LIN {X 0,Y 226.639,Z 302.23,A -85,B 0,C 180,E1 -22455.501,E2 -22455.501} C_VEL
LIN {X 0,Y 230.023,Z 288.136,A -85,B 0,C 180,E1 -22456.446,E2 -22456.446} C_VEL
LIN {X 0,Y 232.529,Z 273.347,A -85,B 0,C 180,E1 -22457.124,E2 -22457.124} C_VEL
LIN {X 0,Y 234.238,Z 254.152,A -85,B 0,C 180,E1 -22457.708,E2 -22457.708} C_VEL
LIN {X 0,Y 236.836,Z 218.214,A -85,B 0,C 180,E1 -22458.708,E2 -22458.708} C_VEL
LIN {X 0,Y 232.194,Z 207.283,A -85,B 0,C 180,E1 -22461.02,E2 -22461.02} C_VEL
LIN {X 0,Y 227.459,Z 197.713,A -85,B 0,C 180,E1 -22463.554,E2 -22463.554} C_VEL
LIN {X 0,Y 222.962,Z 189.346,A -85,B 0,C 180,E1 -22466.218,E2 -22466.218} C_VEL
LIN {X 0,Y 219.708,Z 183.706,A -85,B 0,C 180,E1 -22468.352,E2 -22468.352} C_VEL
LIN {X 0,Y 216.874,Z 179.005,A -85,B 0,C 180,E1 -22470.433,E2 -22470.433} C_VEL
LIN {X 0,Y 214.738,Z 175.538,A -85,B 0,C 180,E1 -22472.178,E2 -22472.178} C_VEL
LIN {X 0,Y 211.845,Z 170.966,A -85,B 0,C 180,E1 -22474.848,E2 -22474.848} C_VEL
LIN {X 0,Y 209.156,Z 167.545,A -85,B 0,C 180,E1 -22477.703,E2 -22477.703} C_VEL
LIN {X 0,Y 207.226,Z 164.238,A -85,B 0,C 180,E1 -22480.325,E2 -22480.325} C_VEL
LIN {X 0,Y 203.698,Z 160.294,A -85,B 0,C 180,E1 -22488.046,E2 -22488.046} C_VEL
LIN {X 0,Y 203.417,Z 158.582,A -85,B 0,C 180,E1 -22490.606,E2 -22490.606} C_VEL
LIN {X 0,Y 203.441,Z 158.596,A -85,B 0,C 180,E1 -22494.045,E2 -22494.045} C_VEL
LIN {X 0,Y 204.542,Z 161.074,A -85,B 0,C 180,E1 -22499.009,E2 -22499.009} C_VEL
LIN {X 0,Y 206.776,Z 163.712,A -85,B 0,C 180,E1 -22503.403,E2 -22503.403} C_VEL
LIN {X 0,Y 207.532,Z 164.297,A -85,B 0,C 180,E1 -22504.485,E2 -22504.485} C_VEL
LIN {X 0,Y 209.461,Z 167.504,A -85,B 0,C 180,E1 -22507.018,E2 -22507.018} C_VEL
LIN {X 0,Y 211.323,Z 169.48,A -85,B 0,C 180,E1 -22508.967,E2 -22508.967} C_VEL
LIN {X 0,Y 213.7,Z 172.996,A -85,B 0,C 180,E1 -22511.242,E2 -22511.242} C_VEL
LIN {X 0,Y 215.003,Z 174.469,A -85,B 0,C 180,E1 -22512.327,E2 -22512.327} C_VEL
LIN {X 0,Y 218.65,Z 179.753,A -85,B 0,C 180,E1 -22515.145,E2 -22515.145} C_VEL
LIN {X 0,Y 221.809,Z 184.298,A -85,B 0,C 180,E1 -22517.251,E2 -22517.251} C_VEL
LIN {X 0,Y 225.031,Z 189.073,A -85,B 0,C 180,E1 -22519.193,E2 -22519.193} C_VEL
LIN {X 0,Y 229.645,Z 196.427,A -85,B 0,C 180,E1 -22521.724,E2 -22521.724} C_VEL
LIN {X 0,Y 234.735,Z 206.452,A -85,B 0,C 180,E1 -22524.318,E2 -22524.318} C_VEL
LIN {X 0,Y 237.283,Z 212.078,A -85,B 0,C 180,E1 -22525.544,E2 -22525.544} C_VEL
LIN {X 0,Y 233.316,Z 263.334,A -85,B 0,C 180,E1 -22526.974,E2 -22526.974} C_VEL
LIN {X 0,Y 231.209,Z 277.512,A -85,B 0,C 180,E1 -22527.622,E2 -22527.622} C_VEL
LIN {X 0,Y 228.377,Z 290.64,A -85,B 0,C 180,E1 -22528.477,E2 -22528.477} C_VEL
LIN {X 0,Y 224.932,Z 303.341,A -85,B 0,C 180,E1 -22529.627,E2 -22529.627} C_VEL
LIN {X 0,Y 220.658,Z 316.029,A -85,B 0,C 180,E1 -22531.128,E2 -22531.128} C_VEL
LIN {X 0,Y 215.677,Z 328.153,A -85,B 0,C 180,E1 -22532.953,E2 -22532.953} C_VEL
LIN {X 0,Y 210.464,Z 339.178,A -85,B 0,C 180,E1 -22535.098,E2 -22535.098} C_VEL
LIN {X 0,Y 205.553,Z 348.32,A -85,B 0,C 180,E1 -22537.347,E2 -22537.347} C_VEL
LIN {X 0,Y 200.034,Z 357.449,A -85,B 0,C 180,E1 -22540.163,E2 -22540.163} C_VEL
LIN {X 0,Y 195.008,Z 365.073,A -85,B 0,C 180,E1 -22543.205,E2 -22543.205} C_VEL
LIN {X 0,Y 190.001,Z 372.031,A -85,B 0,C 180,E1 -22546.816,E2 -22546.816} C_VEL
LIN {X 0,Y 186.208,Z 376.82,A -85,B 0,C 180,E1 -22550.083,E2 -22550.083} C_VEL
LIN {X 0,Y 182.741,Z 380.951,A -85,B 0,C 180,E1 -22553.85,E2 -22553.85} C_VEL
LIN {X 0,Y 180.515,Z 383.439,A -85,B 0,C 180,E1 -22556.967,E2 -22556.967} C_VEL
LIN {X 0,Y 177.978,Z 385.836,A -85,B 0,C 180,E1 -22561.712,E2 -22561.712} C_VEL
LIN {X 0,Y 176.489,Z 386.756,A -85,B 0,C 180,E1 -22566.53,E2 -22566.53} C_VEL
LIN {X 0,Y 175.717,Z 386.244,A -85,B 0,C 180,E1 -22571.336,E2 -22571.336} C_VEL
LIN {X 0,Y 175.641,Z 385.441,A -85,B 0,C 180,E1 -22573.772,E2 -22573.772} C_VEL
LIN {X 0,Y 175.765,Z 382.819,A -85,B 0,C 180,E1 -22578.464,E2 -22578.464} C_VEL
LIN {X 0,Y 176.339,Z 379.84,A -85,B 0,C 180,E1 -22581.978,E2 -22581.978} C_VEL
LIN {X 0,Y 177.183,Z 376.025,A -85,B 0,C 180,E1 -22585.447,E2 -22585.447} C_VEL
LIN {X 0,Y 178.317,Z 371.31,A -85,B 0,C 180,E1 -22588.868,E2 -22588.868} C_VEL
LIN {X 0,Y 180.274,Z 364.443,A -85,B 0,C 180,E1 -22592.79,E2 -22592.79} C_VEL
LIN {X 0,Y 182.883,Z 355.918,A -85,B 0,C 180,E1 -22596.617,E2 -22596.617} C_VEL
LIN {X 0,Y 185.69,Z 346.926,A -85,B 0,C 180,E1 -22599.834,E2 -22599.834} C_VEL
LIN {X 0,Y 188.154,Z 338.243,A -85,B 0,C 180,E1 -22602.399,E2 -22602.399} C_VEL
LIN {X 0,Y 190.884,Z 328.903,A -85,B 0,C 180,E1 -22604.659,E2 -22604.659} C_VEL
LIN {X 0,Y 193.794,Z 317.727,A -85,B 0,C 180,E1 -22606.862,E2 -22606.862} C_VEL
LIN {X 0,Y 196.61,Z 305.55,A -85,B 0,C 180,E1 -22608.763,E2 -22608.763} C_VEL
LIN {X 0,Y 199.157,Z 292.089,A -85,B 0,C 180,E1 -22610.391,E2 -22610.391} C_VEL
LIN {X 0,Y 201.213,Z 278.05,A -85,B 0,C 180,E1 -22611.646,E2 -22611.646} C_VEL
LIN {X 0,Y 202.695,Z 263.821,A -85,B 0,C 180,E1 -22612.518,E2 -22612.518} C_VEL
LIN {X 0,Y 204.368,Z 237.316,A -85,B 0,C 180,E1 -22613.431,E2 -22613.431} C_VEL
LIN {X 0,Y 207.071,Z 187.142,A -85,B 0,C 180,E1 -22615.036,E2 -22615.036} C_VEL
LIN {X 0,Y 202.861,Z 176.015,A -85,B 0,C 180,E1 -22616.361,E2 -22616.361} C_VEL
LIN {X 0,Y 196.456,Z 163.46,A -85,B 0,C 180,E1 -22618.321,E2 -22618.321} C_VEL
LIN {X 0,Y 188.904,Z 150.475,A -85,B 0,C 180,E1 -22620.783,E2 -22620.783} C_VEL
LIN {X 0,Y 183.421,Z 142.139,A -85,B 0,C 180,E1 -22622.704,E2 -22622.704} C_VEL
LIN {X 0,Y 180.927,Z 138.404,A -85,B 0,C 180,E1 -22623.626,E2 -22623.626} C_VEL
LIN {X 0,Y 179.099,Z 136.063,A -85,B 0,C 180,E1 -22624.304,E2 -22624.304} C_VEL
LIN {X 0,Y 178.464,Z 133.88,A -85,B 0,C 180,E1 -22624.658,E2 -22624.658} C_VEL
LIN {X 0,Y 178.477,Z 133.875,A -85,B 0,C 180,E1 -22629.049,E2 -22629.049} C_VEL
LIN {X 0,Y 178.494,Z 133.859,A -85,B 0,C 180,E1 -22632.013,E2 -22632.013} C_VEL
LIN {X 0,Y 178.504,Z 133.854,A -85,B 0,C 180,E1 -22635.123,E2 -22635.123} C_VEL
LIN {X 0,Y 178.493,Z 133.87,A -85,B 0,C 180,E1 -22638.421,E2 -22638.421} C_VEL
LIN {X 0,Y 178.444,Z 133.86,A -85,B 0,C 180,E1 -22643.799,E2 -22643.799} C_VEL
LIN {X 0,Y 178.466,Z 133.878,A -85,B 0,C 180,E1 -22646.553,E2 -22646.553} C_VEL
LIN {X 0,Y 178.499,Z 133.842,A -85,B 0,C 180,E1 -22650.013,E2 -22650.013} C_VEL
LIN {X 0,Y 178.525,Z 133.862,A -85,B 0,C 180,E1 -22654.875,E2 -22654.875} C_VEL
LIN {X 0,Y 178.638,Z 133.852,A -85,B 0,C 180,E1 -22660.761,E2 -22660.761} C_VEL
LIN {X 0,Y 178.663,Z 133.849,A -85,B 0,C 180,E1 -22664.025,E2 -22664.025} C_VEL
LIN {X 0,Y 178.88,Z 133.825,A -85,B 0,C 180,E1 -22669.161,E2 -22669.161} C_VEL
LIN {X 0,Y 178.918,Z 133.782,A -85,B 0,C 180,E1 -22673.24,E2 -22673.24} C_VEL
LIN {X 0,Y 179.146,Z 133.788,A -85,B 0,C 180,E1 -22677.759,E2 -22677.759} C_VEL
LIN {X 0,Y 179.363,Z 133.764,A -85,B 0,C 180,E1 -22680.007,E2 -22680.007} C_VEL
LIN {X 0,Y 178.863,Z 133.791,A -85,B 0,C 180,E1 -22684.515,E2 -22684.515} C_VEL
LIN {X 0,Y 178.953,Z 133.817,A -85,B 0,C 180,E1 -22689.045,E2 -22689.045} C_VEL
LIN {X 0,Y 178.682,Z 133.85,A -85,B 0,C 180,E1 -22693.657,E2 -22693.657} C_VEL
LIN {X 0,Y 178.647,Z 133.853,A -85,B 0,C 180,E1 -22698.351,E2 -22698.351} C_VEL
LIN {X 0,Y 178.51,Z 133.872,A -85,B 0,C 180,E1 -22703.192,E2 -22703.192} C_VEL
LIN {X 0,Y 178.487,Z 133.863,A -85,B 0,C 180,E1 -22708.204,E2 -22708.204} C_VEL
LIN {X 0,Y 178.479,Z 133.872,A -85,B 0,C 180,E1 -22710.798,E2 -22710.798} C_VEL
LIN {X 0,Y 178.486,Z 133.875,A -85,B 0,C 180,E1 -22714.226,E2 -22714.226} C_VEL
LIN {X 0,Y 178.411,Z 134.02,A -85,B 0,C 180,E1 -22719,E2 -22719} C_VEL
LIN {X 0,Y 179.403,Z 136.688,A -85,B 0,C 180,E1 -22719.454,E2 -22719.454} C_VEL
LIN {X 0,Y 181.505,Z 139.246,A -85,B 0,C 180,E1 -22720.224,E2 -22720.224} C_VEL
LIN {X 0,Y 183.847,Z 142.743,A -85,B 0,C 180,E1 -22721.083,E2 -22721.083} C_VEL
LIN {X 0,Y 187.701,Z 149.384,A -85,B 0,C 180,E1 -22722.472,E2 -22722.472} C_VEL
LIN {X 0,Y 194.053,Z 161.878,A -85,B 0,C 180,E1 -22724.674,E2 -22724.674} C_VEL
LIN {X 0,Y 199.515,Z 174.348,A -85,B 0,C 180,E1 -22726.489,E2 -22726.489} C_VEL
LIN {X 0,Y 206.104,Z 192.069,A -85,B 0,C 180,E1 -22728.614,E2 -22728.614} C_VEL
LIN {X 0,Y 206.691,Z 198.413,A -85,B 0,C 180,E1 -22728.996,E2 -22728.996} C_VEL
LIN {X 0,Y 204.55,Z 238.997,A -85,B 0,C 180,E1 -22730.302,E2 -22730.302} C_VEL
LIN {X 0,Y 203.682,Z 244.836,A -85,B 0,C 180,E1 -22730.383,E2 -22730.383} C_VEL
LIN {X 0,Y 197.843,Z 263.771,A -85,B 0,C 180,E1 -22730.101,E2 -22730.101} C_VEL
LIN {X 0,Y 196.93,Z 269.591,A -85,B 0,C 180,E1 -22730.223,E2 -22730.223} C_VEL
LIN {X 0,Y 195.435,Z 283.943,A -85,B 0,C 180,E1 -22731.004,E2 -22731.004} C_VEL
LIN {X 0,Y 193.223,Z 297.885,A -85,B 0,C 180,E1 -22732.14,E2 -22732.14} C_VEL
LIN {X 0,Y 190.752,Z 310.484,A -85,B 0,C 180,E1 -22733.555,E2 -22733.555} C_VEL
LIN {X 0,Y 187.973,Z 322.176,A -85,B 0,C 180,E1 -22735.243,E2 -22735.243} C_VEL
LIN {X 0,Y 184.761,Z 334.344,A -85,B 0,C 180,E1 -22737.505,E2 -22737.505} C_VEL
LIN {X 0,Y 182.676,Z 341.22,A -85,B 0,C 180,E1 -22739.035,E2 -22739.035} C_VEL
LIN {X 0,Y 179.29,Z 352.041,A -85,B 0,C 180,E1 -22741.944,E2 -22741.944} C_VEL
LIN {X 0,Y 176.224,Z 361.794,A -85,B 0,C 180,E1 -22745.248,E2 -22745.248} C_VEL
LIN {X 0,Y 173.711,Z 369.855,A -85,B 0,C 180,E1 -22748.65,E2 -22748.65} C_VEL
LIN {X 0,Y 171.794,Z 376.544,A -85,B 0,C 180,E1 -22752.136,E2 -22752.136} C_VEL
LIN {X 0,Y 170.316,Z 382.067,A -85,B 0,C 180,E1 -22755.669,E2 -22755.669} C_VEL
LIN {X 0,Y 169.282,Z 387.851,A -85,B 0,C 180,E1 -22760.444,E2 -22760.444} C_VEL
LIN {X 0,Y 168.89,Z 392.01,A -85,B 0,C 180,E1 -22765.229,E2 -22765.229} C_VEL
LIN {X 0,Y 169.024,Z 394.686,A -85,B 0,C 180,E1 -22770.003,E2 -22770.003} C_VEL
LIN {X 0,Y 168.891,Z 395.944,A -85,B 0,C 180,E1 -22774.777,E2 -22774.777} C_VEL
LIN {X 0,Y 169.339,Z 395.878,A -85,B 0,C 180,E1 -22779.559,E2 -22779.559} C_VEL
LIN {X 0,Y 170.625,Z 394.512,A -85,B 0,C 180,E1 -22784.312,E2 -22784.312} C_VEL
LIN {X 0,Y 173.086,Z 391.826,A -85,B 0,C 180,E1 -22788.959,E2 -22788.959} C_VEL
LIN {X 0,Y 176.47,Z 387.752,A -85,B 0,C 180,E1 -22793.472,E2 -22793.472} C_VEL
LIN {X 0,Y 180.936,Z 382.174,A -85,B 0,C 180,E1 -22797.785,E2 -22797.785} C_VEL
LIN {X 0,Y 186.475,Z 374.921,A -85,B 0,C 180,E1 -22801.85,E2 -22801.85} C_VEL
LIN {X 0,Y 192.081,Z 366.957,A -85,B 0,C 180,E1 -22805.192,E2 -22805.192} C_VEL
LIN {X 0,Y 197.505,Z 358.65,A -85,B 0,C 180,E1 -22807.87,E2 -22807.87} C_VEL
LIN {X 0,Y 203.298,Z 348.508,A -85,B 0,C 180,E1 -22810.481,E2 -22810.481} C_VEL
LIN {X 0,Y 208.899,Z 337.644,A -85,B 0,C 180,E1 -22812.618,E2 -22812.618} C_VEL
LIN {X 0,Y 214.296,Z 325.305,A -85,B 0,C 180,E1 -22814.511,E2 -22814.511} C_VEL
LIN {X 0,Y 218.855,Z 313.118,A -85,B 0,C 180,E1 -22815.936,E2 -22815.936} C_VEL
LIN {X 0,Y 223.004,Z 299.599,A -85,B 0,C 180,E1 -22817.119,E2 -22817.119} C_VEL
LIN {X 0,Y 226.211,Z 286.174,A -85,B 0,C 180,E1 -22817.967,E2 -22817.967} C_VEL
LIN {X 0,Y 228.574,Z 271.708,A -85,B 0,C 180,E1 -22818.618,E2 -22818.618} C_VEL
LIN {X 0,Y 231.009,Z 242.939,A -85,B 0,C 180,E1 -22819.448,E2 -22819.448} C_VEL
LIN {X 0,Y 232.645,Z 221.01,A -85,B 0,C 180,E1 -22820.066,E2 -22820.066} C_VEL
LIN {X 0,Y 228.436,Z 211.057,A -85,B 0,C 180,E1 -22822.307,E2 -22822.307} C_VEL
LIN {X 0,Y 224.376,Z 202.623,A -85,B 0,C 180,E1 -22824.627,E2 -22824.627} C_VEL
LIN {X 0,Y 220.353,Z 194.856,A -85,B 0,C 180,E1 -22827.16,E2 -22827.16} C_VEL
LIN {X 0,Y 216.306,Z 187.516,A -85,B 0,C 180,E1 -22830.06,E2 -22830.06} C_VEL
LIN {X 0,Y 212.889,Z 181.881,A -85,B 0,C 180,E1 -22832.9,E2 -22832.9} C_VEL
LIN {X 0,Y 209.749,Z 176.823,A -85,B 0,C 180,E1 -22835.99,E2 -22835.99} C_VEL
LIN {X 0,Y 206.06,Z 171.29,A -85,B 0,C 180,E1 -22840.669,E2 -22840.669} C_VEL
LIN {X 0,Y 205.511,Z 170.742,A -85,B 0,C 180,E1 -22841.528,E2 -22841.528} C_VEL
LIN {X 0,Y 202.644,Z 166.883,A -85,B 0,C 180,E1 -22848.997,E2 -22848.997} C_VEL
LIN {X 0,Y 202.501,Z 165.535,A -85,B 0,C 180,E1 -22851.124,E2 -22851.124} C_VEL
LIN {X 0,Y 202.572,Z 165.825,A -85,B 0,C 180,E1 -22854.283,E2 -22854.283} C_VEL
LIN {X 0,Y 203.553,Z 168.062,A -85,B 0,C 180,E1 -22858.757,E2 -22858.757} C_VEL
LIN {X 0,Y 205.721,Z 170.676,A -85,B 0,C 180,E1 -22863.176,E2 -22863.176} C_VEL
LIN {X 0,Y 206.358,Z 171.324,A -85,B 0,C 180,E1 -22864.144,E2 -22864.144} C_VEL
LIN {X 0,Y 208.446,Z 174.671,A -85,B 0,C 180,E1 -22866.938,E2 -22866.938} C_VEL
LIN {X 0,Y 209.825,Z 176.191,A -85,B 0,C 180,E1 -22868.426,E2 -22868.426} C_VEL
LIN {X 0,Y 212.302,Z 179.809,A -85,B 0,C 180,E1 -22870.871,E2 -22870.871} C_VEL
LIN {X 0,Y 213.441,Z 181.322,A -85,B 0,C 180,E1 -22871.869,E2 -22871.869} C_VEL
LIN {X 0,Y 216.66,Z 186.081,A -85,B 0,C 180,E1 -22874.458,E2 -22874.458} C_VEL
LIN {X 0,Y 219.723,Z 190.648,A -85,B 0,C 180,E1 -22876.611,E2 -22876.611} C_VEL
LIN {X 0,Y 223.585,Z 196.497,A -85,B 0,C 180,E1 -22879.006,E2 -22879.006} C_VEL
LIN {X 0,Y 227.202,Z 202.77,A -85,B 0,C 180,E1 -22881.074,E2 -22881.074} C_VEL
LIN {X 0,Y 231.568,Z 211.613,A -85,B 0,C 180,E1 -22883.406,E2 -22883.406} C_VEL
LIN {X 0,Y 233.113,Z 215.025,A -85,B 0,C 180,E1 -22884.192,E2 -22884.192} C_VEL
LIN {X 0,Y 229.221,Z 263.339,A -85,B 0,C 180,E1 -22885.54,E2 -22885.54} C_VEL
LIN {X 0,Y 227.09,Z 277.278,A -85,B 0,C 180,E1 -22886.165,E2 -22886.165} C_VEL
LIN {X 0,Y 223.982,Z 291.266,A -85,B 0,C 180,E1 -22887.08,E2 -22887.08} C_VEL
LIN {X 0,Y 220.076,Z 304.924,A -85,B 0,C 180,E1 -22888.339,E2 -22888.339} C_VEL
LIN {X 0,Y 215.7,Z 317.206,A -85,B 0,C 180,E1 -22889.826,E2 -22889.826} C_VEL
LIN {X 0,Y 210.567,Z 329.156,A -85,B 0,C 180,E1 -22891.664,E2 -22891.664} C_VEL
LIN {X 0,Y 205.077,Z 340.216,A -85,B 0,C 180,E1 -22893.864,E2 -22893.864} C_VEL
LIN {X 0,Y 199.376,Z 350.204,A -85,B 0,C 180,E1 -22896.415,E2 -22896.415} C_VEL
LIN {X 0,Y 193.426,Z 359.414,A -85,B 0,C 180,E1 -22899.453,E2 -22899.453} C_VEL
LIN {X 0,Y 187.543,Z 367.661,A -85,B 0,C 180,E1 -22903.047,E2 -22903.047} C_VEL
LIN {X 0,Y 183.113,Z 373.348,A -85,B 0,C 180,E1 -22906.298,E2 -22906.298} C_VEL
LIN {X 0,Y 179.21,Z 377.935,A -85,B 0,C 180,E1 -22909.675,E2 -22909.675} C_VEL
LIN {X 0,Y 175.978,Z 381.516,A -85,B 0,C 180,E1 -22913.194,E2 -22913.194} C_VEL
LIN {X 0,Y 174.174,Z 383.378,A -85,B 0,C 180,E1 -22915.601,E2 -22915.601} C_VEL
LIN {X 0,Y 171.368,Z 385.895,A -85,B 0,C 180,E1 -22920.515,E2 -22920.515} C_VEL
LIN {X 0,Y 169.591,Z 386.933,A -85,B 0,C 180,E1 -22925.514,E2 -22925.514} C_VEL
LIN {X 0,Y 168.69,Z 386.534,A -85,B 0,C 180,E1 -22930.528,E2 -22930.528} C_VEL
LIN {X 0,Y 168.56,Z 385.64,A -85,B 0,C 180,E1 -22933.496,E2 -22933.496} C_VEL
LIN {X 0,Y 168.611,Z 383.286,A -85,B 0,C 180,E1 -22937.967,E2 -22937.967} C_VEL
LIN {X 0,Y 169.155,Z 380.413,A -85,B 0,C 180,E1 -22941.635,E2 -22941.635} C_VEL
LIN {X 0,Y 170.001,Z 376.719,A -85,B 0,C 180,E1 -22945.254,E2 -22945.254} C_VEL
LIN {X 0,Y 171.156,Z 372.089,A -85,B 0,C 180,E1 -22948.82,E2 -22948.82} C_VEL
LIN {X 0,Y 173.133,Z 365.392,A -85,B 0,C 180,E1 -22952.905,E2 -22952.905} C_VEL
LIN {X 0,Y 175.802,Z 357.048,A -85,B 0,C 180,E1 -22956.885,E2 -22956.885} C_VEL
LIN {X 0,Y 178.897,Z 347.578,A -85,B 0,C 180,E1 -22960.443,E2 -22960.443} C_VEL
LIN {X 0,Y 181.767,Z 337.828,A -85,B 0,C 180,E1 -22963.411,E2 -22963.411} C_VEL
LIN {X 0,Y 184.659,Z 328.358,A -85,B 0,C 180,E1 -22965.731,E2 -22965.731} C_VEL
LIN {X 0,Y 187.72,Z 317.02,A -85,B 0,C 180,E1 -22967.988,E2 -22967.988} C_VEL
LIN {X 0,Y 190.631,Z 304.642,A -85,B 0,C 180,E1 -22969.936,E2 -22969.936} C_VEL
LIN {X 0,Y 193.322,Z 290.861,A -85,B 0,C 180,E1 -22971.594,E2 -22971.594} C_VEL
LIN {X 0,Y 195.335,Z 277.112,A -85,B 0,C 180,E1 -22972.821,E2 -22972.821} C_VEL
LIN {X 0,Y 196.839,Z 262.88,A -85,B 0,C 180,E1 -22973.68,E2 -22973.68} C_VEL
LIN {X 0,Y 200.447,Z 203.666,A -85,B 0,C 180,E1 -22975.643,E2 -22975.643} C_VEL
LIN {X 0,Y 201.212,Z 188.949,A -85,B 0,C 180,E1 -22976.135,E2 -22976.135} C_VEL
LIN {X 0,Y 197.357,Z 178.875,A -85,B 0,C 180,E1 -22977.409,E2 -22977.409} C_VEL
LIN {X 0,Y 191.075,Z 166.594,A -85,B 0,C 180,E1 -22979.443,E2 -22979.443} C_VEL
LIN {X 0,Y 184.097,Z 154.645,A -85,B 0,C 180,E1 -22981.856,E2 -22981.856} C_VEL
LIN {X 0,Y 177.132,Z 143.849,A -85,B 0,C 180,E1 -22984.475,E2 -22984.475} C_VEL
LIN {X 0,Y 174.957,Z 140.891,A -85,B 0,C 180,E1 -22985.334,E2 -22985.334} C_VEL
LIN {X 0,Y 174.114,Z 139.492,A -85,B 0,C 180,E1 -22985.691,E2 -22985.691} C_VEL
LIN {X 0,Y 172.15,Z 137.141,A -85,B 0,C 180,E1 -22986.492,E2 -22986.492} C_VEL
LIN {X 0,Y 171.41,Z 134.76,A -85,B 0,C 180,E1 -22986.954,E2 -22986.954} C_VEL
LIN {X 0,Y 171.434,Z 134.733,A -85,B 0,C 180,E1 -22992.46,E2 -22992.46} C_VEL
LIN {X 0,Y 171.432,Z 134.753,A -85,B 0,C 180,E1 -22997.549,E2 -22997.549} C_VEL
LIN {X 0,Y 171.417,Z 134.721,A -85,B 0,C 180,E1 -23002.06,E2 -23002.06} C_VEL
LIN {X 0,Y 171.395,Z 134.752,A -85,B 0,C 180,E1 -23007.798,E2 -23007.798} C_VEL
LIN {X 0,Y 171.426,Z 134.718,A -85,B 0,C 180,E1 -23010.54,E2 -23010.54} C_VEL
LIN {X 0,Y 171.453,Z 134.75,A -85,B 0,C 180,E1 -23015.81,E2 -23015.81} C_VEL
LIN {X 0,Y 171.594,Z 134.73,A -85,B 0,C 180,E1 -23020.882,E2 -23020.882} C_VEL
LIN {X 0,Y 171.599,Z 134.724,A -85,B 0,C 180,E1 -23025.783,E2 -23025.783} C_VEL
LIN {X 0,Y 171.894,Z 134.682,A -85,B 0,C 180,E1 -23030.596,E2 -23030.596} C_VEL
LIN {X 0,Y 171.814,Z 134.673,A -85,B 0,C 180,E1 -23035.315,E2 -23035.315} C_VEL
LIN {X 0,Y 172.325,Z 134.641,A -85,B 0,C 180,E1 -23040.008,E2 -23040.008} C_VEL
LIN {X 0,Y 171.812,Z 134.668,A -85,B 0,C 180,E1 -23044.7,E2 -23044.7} C_VEL
LIN {X 0,Y 171.883,Z 134.7,A -85,B 0,C 180,E1 -23049.421,E2 -23049.421} C_VEL
LIN {X 0,Y 171.605,Z 134.733,A -85,B 0,C 180,E1 -23054.232,E2 -23054.232} C_VEL
LIN {X 0,Y 171.542,Z 134.742,A -85,B 0,C 180,E1 -23059.57,E2 -23059.57} C_VEL
LIN {X 0,Y 171.469,Z 134.749,A -85,B 0,C 180,E1 -23065.624,E2 -23065.624} C_VEL
LIN {X 0,Y 171.442,Z 134.75,A -85,B 0,C 180,E1 -23070.594,E2 -23070.594} C_VEL
LIN {X 0,Y 171.391,Z 134.759,A -85,B 0,C 180,E1 -23076.674,E2 -23076.674} C_VEL
LIN {X 0,Y 172.273,Z 137.408,A -85,B 0,C 180,E1 -23077.185,E2 -23077.185} C_VEL
LIN {X 0,Y 174.601,Z 140.281,A -85,B 0,C 180,E1 -23078.138,E2 -23078.138} C_VEL
LIN {X 0,Y 176.859,Z 143.654,A -85,B 0,C 180,E1 -23079.056,E2 -23079.056} C_VEL
LIN {X 0,Y 181.273,Z 150.337,A -85,B 0,C 180,E1 -23080.752,E2 -23080.752} C_VEL
LIN {X 0,Y 187.137,Z 161.585,A -85,B 0,C 180,E1 -23082.94,E2 -23082.94} C_VEL
LIN {X 0,Y 193.134,Z 174.722,A -85,B 0,C 180,E1 -23085.065,E2 -23085.065} C_VEL
LIN {X 0,Y 199.773,Z 192.505,A -85,B 0,C 180,E1 -23087.355,E2 -23087.355} C_VEL
LIN {X 0,Y 200.577,Z 195.66,A -85,B 0,C 180,E1 -23087.662,E2 -23087.662} C_VEL
LIN {X 0,Y 200.829,Z 199.802,A -85,B 0,C 180,E1 -23087.896,E2 -23087.896} C_VEL
LIN {X 0,Y 196.93,Z 269.591,A -85,B 0,C 180,E1 -23090.223,E2 -23090.223} C_VEL
LIN {X 0,Y 195.922,Z 275.384,A -85,B 0,C 180,E1 -23090.386,E2 -23090.386} C_VEL
LIN {X 0,Y 192.455,Z 284.667,A -85,B 0,C 180,E1 -23090.492,E2 -23090.492} C_VEL
LIN {X 0,Y 188.566,Z 293.775,A -85,B 0,C 180,E1 -23090.753,E2 -23090.753} C_VEL
LIN {X 0,Y 186.912,Z 299.299,A -85,B 0,C 180,E1 -23091.168,E2 -23091.168} C_VEL
LIN {X 0,Y 184.166,Z 312.3,A -85,B 0,C 180,E1 -23092.717,E2 -23092.717} C_VEL
LIN {X 0,Y 181.138,Z 324.295,A -85,B 0,C 180,E1 -23094.576,E2 -23094.576} C_VEL
LIN {X 0,Y 178.389,Z 334.306,A -85,B 0,C 180,E1 -23096.53,E2 -23096.53} C_VEL
LIN {X 0,Y 176.213,Z 341.167,A -85,B 0,C 180,E1 -23098.103,E2 -23098.103} C_VEL
LIN {X 0,Y 172.993,Z 351.059,A -85,B 0,C 180,E1 -23100.827,E2 -23100.827} C_VEL
LIN {X 0,Y 169.732,Z 360.942,A -85,B 0,C 180,E1 -23104.233,E2 -23104.233} C_VEL
LIN {X 0,Y 166.992,Z 369.253,A -85,B 0,C 180,E1 -23107.819,E2 -23107.819} C_VEL
LIN {X 0,Y 164.703,Z 376.93,A -85,B 0,C 180,E1 -23111.983,E2 -23111.983} C_VEL
LIN {X 0,Y 163.006,Z 383.156,A -85,B 0,C 180,E1 -23116.286,E2 -23116.286} C_VEL
LIN {X 0,Y 162.227,Z 387.382,A -85,B 0,C 180,E1 -23120.025,E2 -23120.025} C_VEL
LIN {X 0,Y 161.946,Z 389.695,A -85,B 0,C 180,E1 -23122.523,E2 -23122.523} C_VEL
LIN {X 0,Y 161.814,Z 393.172,A -85,B 0,C 180,E1 -23127.514,E2 -23127.514} C_VEL
LIN {X 0,Y 161.934,Z 394.368,A -85,B 0,C 180,E1 -23130.004,E2 -23130.004} C_VEL
LIN {X 0,Y 161.81,Z 395.698,A -85,B 0,C 180,E1 -23134.987,E2 -23134.987} C_VEL
LIN {X 0,Y 162.326,Z 395.706,A -85,B 0,C 180,E1 -23139.976,E2 -23139.976} C_VEL
LIN {X 0,Y 163.709,Z 394.42,A -85,B 0,C 180,E1 -23144.93,E2 -23144.93} C_VEL
LIN {X 0,Y 166.338,Z 391.824,A -85,B 0,C 180,E1 -23149.759,E2 -23149.759} C_VEL
LIN {X 0,Y 169.94,Z 387.837,A -85,B 0,C 180,E1 -23154.432,E2 -23154.432} C_VEL
LIN {X 0,Y 174.677,Z 382.342,A -85,B 0,C 180,E1 -23158.873,E2 -23158.873} C_VEL
LIN {X 0,Y 180.486,Z 375.178,A -85,B 0,C 180,E1 -23163.038,E2 -23163.038} C_VEL
LIN {X 0,Y 186.339,Z 367.314,A -85,B 0,C 180,E1 -23166.447,E2 -23166.447} C_VEL
LIN {X 0,Y 191.977,Z 359.12,A -85,B 0,C 180,E1 -23169.164,E2 -23169.164} C_VEL
LIN {X 0,Y 197.774,Z 349.473,A -85,B 0,C 180,E1 -23171.726,E2 -23171.726} C_VEL
LIN {X 0,Y 203.779,Z 338.449,A -85,B 0,C 180,E1 -23173.957,E2 -23173.957} C_VEL
LIN {X 0,Y 209.345,Z 326.429,A -85,B 0,C 180,E1 -23175.859,E2 -23175.859} C_VEL
LIN {X 0,Y 214.042,Z 314.572,A -85,B 0,C 180,E1 -23177.283,E2 -23177.283} C_VEL
LIN {X 0,Y 218.273,Z 301.536,A -85,B 0,C 180,E1 -23178.474,E2 -23178.474} C_VEL
LIN {X 0,Y 221.878,Z 287.347,A -85,B 0,C 180,E1 -23179.398,E2 -23179.398} C_VEL
LIN {X 0,Y 224.442,Z 272.737,A -85,B 0,C 180,E1 -23180.066,E2 -23180.066} C_VEL
LIN {X 0,Y 226.373,Z 252.123,A -85,B 0,C 180,E1 -23180.688,E2 -23180.688} C_VEL
LIN {X 0,Y 228.588,Z 223.962,A -85,B 0,C 180,E1 -23181.469,E2 -23181.469} C_VEL
LIN {X 0,Y 225.133,Z 215.618,A -85,B 0,C 180,E1 -23183.437,E2 -23183.437} C_VEL
LIN {X 0,Y 221.106,Z 206.893,A -85,B 0,C 180,E1 -23185.908,E2 -23185.908} C_VEL
LIN {X 0,Y 217.495,Z 199.828,A -85,B 0,C 180,E1 -23188.341,E2 -23188.341} C_VEL
LIN {X 0,Y 213.873,Z 193.038,A -85,B 0,C 180,E1 -23191.153,E2 -23191.153} C_VEL
LIN {X 0,Y 211.177,Z 188.352,A -85,B 0,C 180,E1 -23193.54,E2 -23193.54} C_VEL
LIN {X 0,Y 208.172,Z 183.358,A -85,B 0,C 180,E1 -23196.654,E2 -23196.654} C_VEL
LIN {X 0,Y 204.661,Z 177.829,A -85,B 0,C 180,E1 -23201.448,E2 -23201.448} C_VEL
LIN {X 0,Y 201.755,Z 174.043,A -85,B 0,C 180,E1 -23208.948,E2 -23208.948} C_VEL
LIN {X 0,Y 201.611,Z 172.649,A -85,B 0,C 180,E1 -23211.085,E2 -23211.085} C_VEL
LIN {X 0,Y 201.658,Z 172.794,A -85,B 0,C 180,E1 -23213.992,E2 -23213.992} C_VEL
LIN {X 0,Y 202.581,Z 175.069,A -85,B 0,C 180,E1 -23218.548,E2 -23218.548} C_VEL
LIN {X 0,Y 204.668,Z 177.649,A -85,B 0,C 180,E1 -23222.946,E2 -23222.946} C_VEL
LIN {X 0,Y 205.196,Z 178.331,A -85,B 0,C 180,E1 -23223.798,E2 -23223.798} C_VEL
LIN {X 0,Y 207.332,Z 181.654,A -85,B 0,C 180,E1 -23226.731,E2 -23226.731} C_VEL
LIN {X 0,Y 208.445,Z 183.081,A -85,B 0,C 180,E1 -23227.99,E2 -23227.99} C_VEL
LIN {X 0,Y 211.139,Z 186.884,A -85,B 0,C 180,E1 -23230.699,E2 -23230.699} C_VEL
LIN {X 0,Y 214.733,Z 192.434,A -85,B 0,C 180,E1 -23233.78,E2 -23233.78} C_VEL
LIN {X 0,Y 218.372,Z 197.995,A -85,B 0,C 180,E1 -23236.43,E2 -23236.43} C_VEL
LIN {X 0,Y 223.043,Z 205.661,A -85,B 0,C 180,E1 -23239.37,E2 -23239.37} C_VEL
LIN {X 0,Y 227.705,Z 214.964,A -85,B 0,C 180,E1 -23242.046,E2 -23242.046} C_VEL
LIN {X 0,Y 229.029,Z 218.048,A -85,B 0,C 180,E1 -23242.776,E2 -23242.776} C_VEL
LIN {X 0,Y 225.192,Z 264.021,A -85,B 0,C 180,E1 -23244.078,E2 -23244.078} C_VEL
LIN {X 0,Y 222.937,Z 278.157,A -85,B 0,C 180,E1 -23244.723,E2 -23244.723} C_VEL
LIN {X 0,Y 220.032,Z 290.765,A -85,B 0,C 180,E1 -23245.529,E2 -23245.529} C_VEL
LIN {X 0,Y 216.315,Z 303.617,A -85,B 0,C 180,E1 -23246.685,E2 -23246.685} C_VEL
LIN {X 0,Y 211.464,Z 316.962,A -85,B 0,C 180,E1 -23248.265,E2 -23248.265} C_VEL
LIN {X 0,Y 206.151,Z 328.977,A -85,B 0,C 180,E1 -23250.104,E2 -23250.104} C_VEL
LIN {X 0,Y 200.765,Z 339.423,A -85,B 0,C 180,E1 -23252.154,E2 -23252.154} C_VEL
LIN {X 0,Y 194.809,Z 349.606,A -85,B 0,C 180,E1 -23254.716,E2 -23254.716} C_VEL
LIN {X 0,Y 188.689,Z 358.735,A -85,B 0,C 180,E1 -23257.671,E2 -23257.671} C_VEL
LIN {X 0,Y 183.639,Z 365.658,A -85,B 0,C 180,E1 -23260.576,E2 -23260.576} C_VEL
LIN {X 0,Y 179.21,Z 371.154,A -85,B 0,C 180,E1 -23263.485,E2 -23263.485} C_VEL
LIN {X 0,Y 174.838,Z 376.209,A -85,B 0,C 180,E1 -23266.89,E2 -23266.89} C_VEL
LIN {X 0,Y 171.065,Z 380.235,A -85,B 0,C 180,E1 -23270.443,E2 -23270.443} C_VEL
LIN {X 0,Y 167.941,Z 383.278,A -85,B 0,C 180,E1 -23274.131,E2 -23274.131} C_VEL
LIN {X 0,Y 165.347,Z 385.525,A -85,B 0,C 180,E1 -23278.203,E2 -23278.203} C_VEL
LIN {X 0,Y 163.651,Z 386.716,A -85,B 0,C 180,E1 -23281.806,E2 -23281.806} C_VEL
LIN {X 0,Y 162.113,Z 387.145,A -85,B 0,C 180,E1 -23287.031,E2 -23287.031} C_VEL
LIN {X 0,Y 161.478,Z 386.148,A -85,B 0,C 180,E1 -23292.259,E2 -23292.259} C_VEL
LIN {X 0,Y 161.414,Z 385.121,A -85,B 0,C 180,E1 -23294.853,E2 -23294.853} C_VEL
LIN {X 0,Y 161.769,Z 382.001,A -85,B 0,C 180,E1 -23299.989,E2 -23299.989} C_VEL
LIN {X 0,Y 162.538,Z 378.564,A -85,B 0,C 180,E1 -23303.893,E2 -23303.893} C_VEL
LIN {X 0,Y 163.976,Z 372.847,A -85,B 0,C 180,E1 -23308.769,E2 -23308.769} C_VEL
LIN {X 0,Y 165.978,Z 366.288,A -85,B 0,C 180,E1 -23313.031,E2 -23313.031} C_VEL
LIN {X 0,Y 168.723,Z 358.15,A -85,B 0,C 180,E1 -23317.175,E2 -23317.175} C_VEL
LIN {X 0,Y 171.458,Z 350.198,A -85,B 0,C 180,E1 -23320.396,E2 -23320.396} C_VEL
LIN {X 0,Y 174.337,Z 341.181,A -85,B 0,C 180,E1 -23323.399,E2 -23323.399} C_VEL
LIN {X 0,Y 177.381,Z 331.208,A -85,B 0,C 180,E1 -23326.098,E2 -23326.098} C_VEL
LIN {X 0,Y 180.594,Z 320.401,A -85,B 0,C 180,E1 -23328.429,E2 -23328.429} C_VEL
LIN {X 0,Y 183.631,Z 308.759,A -85,B 0,C 180,E1 -23330.437,E2 -23330.437} C_VEL
LIN {X 0,Y 186.548,Z 295.148,A -85,B 0,C 180,E1 -23332.274,E2 -23332.274} C_VEL
LIN {X 0,Y 188.76,Z 282.081,A -85,B 0,C 180,E1 -23333.59,E2 -23333.59} C_VEL
LIN {X 0,Y 190.46,Z 268.088,A -85,B 0,C 180,E1 -23334.596,E2 -23334.596} C_VEL
LIN {X 0,Y 191.662,Z 253.444,A -85,B 0,C 180,E1 -23335.228,E2 -23335.228} C_VEL
LIN {X 0,Y 195.398,Z 190.619,A -85,B 0,C 180,E1 -23337.304,E2 -23337.304} C_VEL
LIN {X 0,Y 192.258,Z 182.569,A -85,B 0,C 180,E1 -23338.394,E2 -23338.394} C_VEL
LIN {X 0,Y 186.411,Z 170.947,A -85,B 0,C 180,E1 -23340.402,E2 -23340.402} C_VEL
LIN {X 0,Y 179.803,Z 159.387,A -85,B 0,C 180,E1 -23342.819,E2 -23342.819} C_VEL
LIN {X 0,Y 173.098,Z 148.974,A -85,B 0,C 180,E1 -23345.472,E2 -23345.472} C_VEL
LIN {X 0,Y 169.895,Z 144.445,A -85,B 0,C 180,E1 -23346.833,E2 -23346.833} C_VEL
LIN {X 0,Y 167.685,Z 140.987,A -85,B 0,C 180,E1 -23347.845,E2 -23347.845} C_VEL
LIN {X 0,Y 165.205,Z 138.17,A -85,B 0,C 180,E1 -23348.967,E2 -23348.967} C_VEL
LIN {X 0,Y 164.377,Z 135.633,A -85,B 0,C 180,E1 -23349.532,E2 -23349.532} C_VEL
LIN {X 0,Y 164.367,Z 135.607,A -85,B 0,C 180,E1 -23353.388,E2 -23353.388} C_VEL
LIN {X 0,Y 164.371,Z 135.63,A -85,B 0,C 180,E1 -23356.847,E2 -23356.847} C_VEL
LIN {X 0,Y 164.352,Z 135.607,A -85,B 0,C 180,E1 -23360.322,E2 -23360.322} C_VEL
LIN {X 0,Y 164.324,Z 135.623,A -85,B 0,C 180,E1 -23364.346,E2 -23364.346} C_VEL
LIN {X 0,Y 164.367,Z 135.61,A -85,B 0,C 180,E1 -23369.14,E2 -23369.14} C_VEL
LIN {X 0,Y 164.404,Z 135.617,A -85,B 0,C 180,E1 -23374.702,E2 -23374.702} C_VEL
LIN {X 0,Y 164.502,Z 135.609,A -85,B 0,C 180,E1 -23380.024,E2 -23380.024} C_VEL
LIN {X 0,Y 164.546,Z 135.602,A -85,B 0,C 180,E1 -23385.16,E2 -23385.16} C_VEL
LIN {X 0,Y 164.837,Z 135.565,A -85,B 0,C 180,E1 -23390.189,E2 -23390.189} C_VEL
LIN {X 0,Y 164.763,Z 135.547,A -85,B 0,C 180,E1 -23395.114,E2 -23395.114} C_VEL
LIN {X 0,Y 165.287,Z 135.518,A -85,B 0,C 180,E1 -23400.008,E2 -23400.008} C_VEL
LIN {X 0,Y 164.762,Z 135.545,A -85,B 0,C 180,E1 -23404.902,E2 -23404.902} C_VEL
LIN {X 0,Y 164.844,Z 135.558,A -85,B 0,C 180,E1 -23407.356,E2 -23407.356} C_VEL
LIN {X 0,Y 164.748,Z 135.583,A -85,B 0,C 180,E1 -23411.16,E2 -23411.16} C_VEL
LIN {X 0,Y 164.502,Z 135.611,A -85,B 0,C 180,E1 -23417.409,E2 -23417.409} C_VEL
LIN {X 0,Y 164.471,Z 135.623,A -85,B 0,C 180,E1 -23419.997,E2 -23419.997} C_VEL
LIN {X 0,Y 164.393,Z 135.626,A -85,B 0,C 180,E1 -23426.142,E2 -23426.142} C_VEL
LIN {X 0,Y 164.376,Z 135.626,A -85,B 0,C 180,E1 -23431.235,E2 -23431.235} C_VEL
LIN {X 0,Y 164.334,Z 135.731,A -85,B 0,C 180,E1 -23434.147,E2 -23434.147} C_VEL
LIN {X 0,Y 165.151,Z 138.154,A -85,B 0,C 180,E1 -23434.626,E2 -23434.626} C_VEL
LIN {X 0,Y 167.212,Z 140.507,A -85,B 0,C 180,E1 -23435.563,E2 -23435.563} C_VEL
LIN {X 0,Y 170.151,Z 144.786,A -85,B 0,C 180,E1 -23436.893,E2 -23436.893} C_VEL
LIN {X 0,Y 176.242,Z 153.813,A -85,B 0,C 180,E1 -23439.436,E2 -23439.436} C_VEL
LIN {X 0,Y 179.678,Z 160.01,A -85,B 0,C 180,E1 -23440.811,E2 -23440.811} C_VEL
LIN {X 0,Y 186.476,Z 174.512,A -85,B 0,C 180,E1 -23443.419,E2 -23443.419} C_VEL
LIN {X 0,Y 191.641,Z 187.698,A -85,B 0,C 180,E1 -23445.33,E2 -23445.33} C_VEL
LIN {X 0,Y 194.904,Z 197.329,A -85,B 0,C 180,E1 -23446.525,E2 -23446.525} C_VEL
LIN {X 0,Y 194.94,Z 202.481,A -85,B 0,C 180,E1 -23446.77,E2 -23446.77} C_VEL
LIN {X 0,Y 190.927,Z 271.064,A -85,B 0,C 180,E1 -23449.121,E2 -23449.121} C_VEL
LIN {X 0,Y 189.24,Z 285.698,A -85,B 0,C 180,E1 -23449.992,E2 -23449.992} C_VEL
LIN {X 0,Y 186.912,Z 299.299,A -85,B 0,C 180,E1 -23451.168,E2 -23451.168} C_VEL
LIN {X 0,Y 185.171,Z 304.797,A -85,B 0,C 180,E1 -23451.643,E2 -23451.643} C_VEL
LIN {X 0,Y 180.745,Z 313.407,A -85,B 0,C 180,E1 -23452.283,E2 -23452.283} C_VEL
LIN {X 0,Y 176.183,Z 321.781,A -85,B 0,C 180,E1 -23453.134,E2 -23453.134} C_VEL
LIN {X 0,Y 174.268,Z 326.774,A -85,B 0,C 180,E1 -23453.944,E2 -23453.944} C_VEL
LIN {X 0,Y 171.644,Z 335.412,A -85,B 0,C 180,E1 -23455.741,E2 -23455.741} C_VEL
LIN {X 0,Y 168.826,Z 344.268,A -85,B 0,C 180,E1 -23457.947,E2 -23457.947} C_VEL
LIN {X 0,Y 164.935,Z 355.301,A -85,B 0,C 180,E1 -23461.36,E2 -23461.36} C_VEL
LIN {X 0,Y 161.773,Z 364.409,A -85,B 0,C 180,E1 -23464.944,E2 -23464.944} C_VEL
LIN {X 0,Y 159.266,Z 371.711,A -85,B 0,C 180,E1 -23468.505,E2 -23468.505} C_VEL
LIN {X 0,Y 157.613,Z 377.307,A -85,B 0,C 180,E1 -23471.816,E2 -23471.816} C_VEL
LIN {X 0,Y 156.049,Z 382.598,A -85,B 0,C 180,E1 -23475.662,E2 -23475.662} C_VEL
LIN {X 0,Y 155.032,Z 388.168,A -85,B 0,C 180,E1 -23480.874,E2 -23480.874} C_VEL
LIN {X 0,Y 154.724,Z 391.226,A -85,B 0,C 180,E1 -23484.792,E2 -23484.792} C_VEL
LIN {X 0,Y 154.729,Z 393.142,A -85,B 0,C 180,E1 -23487.987,E2 -23487.987} C_VEL
LIN {X 0,Y 154.835,Z 394.047,A -85,B 0,C 180,E1 -23490.004,E2 -23490.004} C_VEL
LIN {X 0,Y 154.725,Z 395.448,A -85,B 0,C 180,E1 -23495.216,E2 -23495.216} C_VEL
LIN {X 0,Y 155.298,Z 395.527,A -85,B 0,C 180,E1 -23500.433,E2 -23500.433} C_VEL
LIN {X 0,Y 156.816,Z 394.313,A -85,B 0,C 180,E1 -23505.603,E2 -23505.603} C_VEL
LIN {X 0,Y 159.628,Z 391.797,A -85,B 0,C 180,E1 -23510.627,E2 -23510.627} C_VEL
LIN {X 0,Y 163.487,Z 387.911,A -85,B 0,C 180,E1 -23515.464,E2 -23515.464} C_VEL
LIN {X 0,Y 168.471,Z 382.51,A -85,B 0,C 180,E1 -23520.043,E2 -23520.043} C_VEL
LIN {X 0,Y 174.566,Z 375.443,A -85,B 0,C 180,E1 -23524.311,E2 -23524.311} C_VEL
LIN {X 0,Y 180.698,Z 367.692,A -85,B 0,C 180,E1 -23527.78,E2 -23527.78} C_VEL
LIN {X 0,Y 186.552,Z 359.628,A -85,B 0,C 180,E1 -23530.535,E2 -23530.535} C_VEL
LIN {X 0,Y 192.865,Z 349.635,A -85,B 0,C 180,E1 -23533.237,E2 -23533.237} C_VEL
LIN {X 0,Y 199.321,Z 338.21,A -85,B 0,C 180,E1 -23535.566,E2 -23535.566} C_VEL
LIN {X 0,Y 205.112,Z 326.173,A -85,B 0,C 180,E1 -23537.453,E2 -23537.453} C_VEL
LIN {X 0,Y 209.955,Z 314.303,A -85,B 0,C 180,E1 -23538.869,E2 -23538.869} C_VEL
LIN {X 0,Y 214.33,Z 301.236,A -85,B 0,C 180,E1 -23540.043,E2 -23540.043} C_VEL
LIN {X 0,Y 218.062,Z 286.937,A -85,B 0,C 180,E1 -23540.955,E2 -23540.955} C_VEL
LIN {X 0,Y 220.694,Z 272.118,A -85,B 0,C 180,E1 -23541.628,E2 -23541.628} C_VEL
LIN {X 0,Y 222.743,Z 250.64,A -85,B 0,C 180,E1 -23542.263,E2 -23542.263} C_VEL
LIN {X 0,Y 224.69,Z 226.904,A -85,B 0,C 180,E1 -23542.915,E2 -23542.915} C_VEL
LIN {X 0,Y 220.725,Z 217.299,A -85,B 0,C 180,E1 -23545.369,E2 -23545.369} C_VEL
LIN {X 0,Y 216.281,Z 207.768,A -85,B 0,C 180,E1 -23548.405,E2 -23548.405} C_VEL
LIN {X 0,Y 212.147,Z 199.622,A -85,B 0,C 180,E1 -23551.726,E2 -23551.726} C_VEL
LIN {X 0,Y 209.361,Z 194.613,A -85,B 0,C 180,E1 -23554.321,E2 -23554.321} C_VEL
LIN {X 0,Y 206.557,Z 189.777,A -85,B 0,C 180,E1 -23557.407,E2 -23557.407} C_VEL
LIN {X 0,Y 203.483,Z 184.732,A -85,B 0,C 180,E1 -23561.884,E2 -23561.884} C_VEL
LIN {X 0,Y 200.773,Z 180.763,A -85,B 0,C 180,E1 -23569.659,E2 -23569.659} C_VEL
LIN {X 0,Y 200.704,Z 179.643,A -85,B 0,C 180,E1 -23571.493,E2 -23571.493} C_VEL
LIN {X 0,Y 200.759,Z 179.928,A -85,B 0,C 180,E1 -23573.965,E2 -23573.965} C_VEL
LIN {X 0,Y 201.566,Z 181.948,A -85,B 0,C 180,E1 -23578.177,E2 -23578.177} C_VEL
LIN {X 0,Y 203.62,Z 184.599,A -85,B 0,C 180,E1 -23582.712,E2 -23582.712} C_VEL
LIN {X 0,Y 204.402,Z 186.063,A -85,B 0,C 180,E1 -23584.06,E2 -23584.06} C_VEL
LIN {X 0,Y 207.049,Z 189.846,A -85,B 0,C 180,E1 -23587.507,E2 -23587.507} C_VEL
LIN {X 0,Y 210.239,Z 194.669,A -85,B 0,C 180,E1 -23590.804,E2 -23590.804} C_VEL
LIN {X 0,Y 212.869,Z 198.792,A -85,B 0,C 180,E1 -23593.113,E2 -23593.113} C_VEL
LIN {X 0,Y 216.867,Z 205.161,A -85,B 0,C 180,E1 -23596.145,E2 -23596.145} C_VEL
LIN {X 0,Y 221.327,Z 212.992,A -85,B 0,C 180,E1 -23599.048,E2 -23599.048} C_VEL
LIN {X 0,Y 225.14,Z 221.282,A -85,B 0,C 180,E1 -23601.345,E2 -23601.345} C_VEL
LIN {X 0,Y 221.364,Z 264.336,A -85,B 0,C 180,E1 -23602.548,E2 -23602.548} C_VEL
LIN {X 0,Y 218.914,Z 279.016,A -85,B 0,C 180,E1 -23603.218,E2 -23603.218} C_VEL
LIN {X 0,Y 215.934,Z 291.46,A -85,B 0,C 180,E1 -23604.022,E2 -23604.022} C_VEL
LIN {X 0,Y 212.414,Z 303.261,A -85,B 0,C 180,E1 -23605.071,E2 -23605.071} C_VEL
LIN {X 0,Y 207.902,Z 315.501,A -85,B 0,C 180,E1 -23606.482,E2 -23606.482} C_VEL
LIN {X 0,Y 202.485,Z 327.576,A -85,B 0,C 180,E1 -23608.264,E2 -23608.264} C_VEL
LIN {X 0,Y 196.658,Z 338.661,A -85,B 0,C 180,E1 -23610.379,E2 -23610.379} C_VEL
LIN {X 0,Y 190.477,Z 348.925,A -85,B 0,C 180,E1 -23612.919,E2 -23612.919} C_VEL
LIN {X 0,Y 184.171,Z 358.033,A -85,B 0,C 180,E1 -23615.811,E2 -23615.811} C_VEL
LIN {X 0,Y 178.065,Z 366.003,A -85,B 0,C 180,E1 -23619.15,E2 -23619.15} C_VEL
LIN {X 0,Y 172.438,Z 372.599,A -85,B 0,C 180,E1 -23622.805,E2 -23622.805} C_VEL
LIN {X 0,Y 167.922,Z 377.389,A -85,B 0,C 180,E1 -23626.32,E2 -23626.32} C_VEL
LIN {X 0,Y 163.411,Z 381.78,A -85,B 0,C 180,E1 -23630.712,E2 -23630.712} C_VEL
LIN {X 0,Y 159.956,Z 384.766,A -85,B 0,C 180,E1 -23635.163,E2 -23635.163} C_VEL
LIN {X 0,Y 157.016,Z 386.825,A -85,B 0,C 180,E1 -23640.5,E2 -23640.5} C_VEL
LIN {X 0,Y 155.23,Z 387.379,A -85,B 0,C 180,E1 -23645.95,E2 -23645.95} C_VEL
LIN {X 0,Y 154.433,Z 386.492,A -85,B 0,C 180,E1 -23651.42,E2 -23651.42} C_VEL
LIN {X 0,Y 154.339,Z 385.518,A -85,B 0,C 180,E1 -23654.141,E2 -23654.141} C_VEL
LIN {X 0,Y 154.579,Z 382.511,A -85,B 0,C 180,E1 -23659.518,E2 -23659.518} C_VEL
LIN {X 0,Y 155.438,Z 378.809,A -85,B 0,C 180,E1 -23664.003,E2 -23664.003} C_VEL
LIN {X 0,Y 156.803,Z 373.593,A -85,B 0,C 180,E1 -23668.712,E2 -23668.712} C_VEL
LIN {X 0,Y 158.828,Z 367.169,A -85,B 0,C 180,E1 -23673.167,E2 -23673.167} C_VEL
LIN {X 0,Y 161.651,Z 359.176,A -85,B 0,C 180,E1 -23677.491,E2 -23677.491} C_VEL
LIN {X 0,Y 164.911,Z 350.124,A -85,B 0,C 180,E1 -23681.341,E2 -23681.341} C_VEL
LIN {X 0,Y 168.005,Z 340.788,A -85,B 0,C 180,E1 -23684.533,E2 -23684.533} C_VEL
LIN {X 0,Y 170.897,Z 331.765,A -85,B 0,C 180,E1 -23687.035,E2 -23687.035} C_VEL
LIN {X 0,Y 174.235,Z 321.032,A -85,B 0,C 180,E1 -23689.434,E2 -23689.434} C_VEL
LIN {X 0,Y 177.793,Z 307.903,A -85,B 0,C 180,E1 -23691.748,E2 -23691.748} C_VEL
LIN {X 0,Y 180.63,Z 295.018,A -85,B 0,C 180,E1 -23693.5,E2 -23693.5} C_VEL
LIN {X 0,Y 183.025,Z 281.106,A -85,B 0,C 180,E1 -23694.906,E2 -23694.906} C_VEL
LIN {X 0,Y 184.816,Z 266.429,A -85,B 0,C 180,E1 -23695.929,E2 -23695.929} C_VEL
LIN {X 0,Y 186.059,Z 250.771,A -85,B 0,C 180,E1 -23696.572,E2 -23696.572} C_VEL
LIN {X 0,Y 189.711,Z 192.551,A -85,B 0,C 180,E1 -23698.519,E2 -23698.519} C_VEL
LIN {X 0,Y 186.693,Z 185.07,A -85,B 0,C 180,E1 -23699.624,E2 -23699.624} C_VEL
LIN {X 0,Y 180.33,Z 172.464,A -85,B 0,C 180,E1 -23701.969,E2 -23701.969} C_VEL
LIN {X 0,Y 173.877,Z 161.345,A -85,B 0,C 180,E1 -23704.503,E2 -23704.503} C_VEL
LIN {X 0,Y 168.485,Z 153.177,A -85,B 0,C 180,E1 -23706.795,E2 -23706.795} C_VEL
LIN {X 0,Y 166.15,Z 149.74,A -85,B 0,C 180,E1 -23707.86,E2 -23707.86} C_VEL
LIN {X 0,Y 163.658,Z 146.027,A -85,B 0,C 180,E1 -23709.057,E2 -23709.057} C_VEL
LIN {X 0,Y 161.372,Z 143.032,A -85,B 0,C 180,E1 -23710.186,E2 -23710.186} C_VEL
LIN {X 0,Y 160.594,Z 141.677,A -85,B 0,C 180,E1 -23710.607,E2 -23710.607} C_VEL
LIN {X 0,Y 158.312,Z 139.434,A -85,B 0,C 180,E1 -23711.764,E2 -23711.764} C_VEL
LIN {X 0,Y 157.313,Z 136.739,A -85,B 0,C 180,E1 -23712.416,E2 -23712.416} C_VEL
LIN {X 0,Y 157.297,Z 136.491,A -85,B 0,C 180,E1 -23712.514,E2 -23712.514} C_VEL
LIN {X 0,Y 157.271,Z 136.517,A -85,B 0,C 180,E1 -23717.922,E2 -23717.922} C_VEL
LIN {X 0,Y 157.301,Z 136.485,A -85,B 0,C 180,E1 -23723.528,E2 -23723.528} C_VEL
LIN {X 0,Y 157.271,Z 136.508,A -85,B 0,C 180,E1 -23728.102,E2 -23728.102} C_VEL
LIN {X 0,Y 157.305,Z 136.482,A -85,B 0,C 180,E1 -23733.473,E2 -23733.473} C_VEL
LIN {X 0,Y 157.429,Z 136.489,A -85,B 0,C 180,E1 -23739.623,E2 -23739.623} C_VEL
LIN {X 0,Y 157.474,Z 136.485,A -85,B 0,C 180,E1 -23744.477,E2 -23744.477} C_VEL
LIN {X 0,Y 157.757,Z 136.45,A -85,B 0,C 180,E1 -23749.744,E2 -23749.744} C_VEL
LIN {X 0,Y 157.809,Z 136.411,A -85,B 0,C 180,E1 -23752.331,E2 -23752.331} C_VEL
LIN {X 0,Y 158.249,Z 136.394,A -85,B 0,C 180,E1 -23760.008,E2 -23760.008} C_VEL
LIN {X 0,Y 157.802,Z 136.438,A -85,B 0,C 180,E1 -23767.686,E2 -23767.686} C_VEL
LIN {X 0,Y 157.678,Z 136.463,A -85,B 0,C 180,E1 -23771.33,E2 -23771.33} C_VEL
LIN {X 0,Y 157.474,Z 136.493,A -85,B 0,C 180,E1 -23775.54,E2 -23775.54} C_VEL
LIN {X 0,Y 157.368,Z 136.504,A -85,B 0,C 180,E1 -23780.941,E2 -23780.941} C_VEL
LIN {X 0,Y 157.314,Z 136.503,A -85,B 0,C 180,E1 -23786.693,E2 -23786.693} C_VEL
LIN {X 0,Y 157.359,Z 136.499,A -85,B 0,C 180,E1 -23791.196,E2 -23791.196} C_VEL
LIN {X 0,Y 158.146,Z 139.101,A -85,B 0,C 180,E1 -23791.771,E2 -23791.771} C_VEL
LIN {X 0,Y 160.016,Z 141.285,A -85,B 0,C 180,E1 -23792.745,E2 -23792.745} C_VEL
LIN {X 0,Y 160.917,Z 142.2,A -85,B 0,C 180,E1 -23793.19,E2 -23793.19} C_VEL
LIN {X 0,Y 163.097,Z 145.539,A -85,B 0,C 180,E1 -23794.306,E2 -23794.306} C_VEL
LIN {X 0,Y 164.461,Z 147.244,A -85,B 0,C 180,E1 -23794.953,E2 -23794.953} C_VEL
LIN {X 0,Y 171.828,Z 158.11,A -85,B 0,C 180,E1 -23798.265,E2 -23798.265} C_VEL
LIN {X 0,Y 175.525,Z 165.073,A -85,B 0,C 180,E1 -23799.847,E2 -23799.847} C_VEL
LIN {X 0,Y 181.579,Z 178.258,A -85,B 0,C 180,E1 -23802.315,E2 -23802.315} C_VEL
LIN {X 0,Y 186.446,Z 190.92,A -85,B 0,C 180,E1 -23804.231,E2 -23804.231} C_VEL
LIN {X 0,Y 189.407,Z 199.683,A -85,B 0,C 180,E1 -23805.378,E2 -23805.378} C_VEL
LIN {X 0,Y 185.076,Z 271.3,A -85,B 0,C 180,E1 -23807.901,E2 -23807.901} C_VEL
LIN {X 0,Y 183.329,Z 285.793,A -85,B 0,C 180,E1 -23808.789,E2 -23808.789} C_VEL
LIN {X 0,Y 180.925,Z 299.293,A -85,B 0,C 180,E1 -23809.985,E2 -23809.985} C_VEL
LIN {X 0,Y 178.079,Z 312.277,A -85,B 0,C 180,E1 -23811.572,E2 -23811.572} C_VEL
LIN {X 0,Y 174.864,Z 324.428,A -85,B 0,C 180,E1 -23813.507,E2 -23813.507} C_VEL
LIN {X 0,Y 174.268,Z 326.774,A -85,B 0,C 180,E1 -23813.944,E2 -23813.944} C_VEL
LIN {X 0,Y 172.726,Z 330.066,A -85,B 0,C 180,E1 -23814.493,E2 -23814.493} C_VEL
LIN {X 0,Y 168.602,Z 335.097,A -85,B 0,C 180,E1 -23815.131,E2 -23815.131} C_VEL
LIN {X 0,Y 164.417,Z 339.982,A -85,B 0,C 180,E1 -23815.86,E2 -23815.86} C_VEL
LIN {X 0,Y 162.796,Z 342.999,A -85,B 0,C 180,E1 -23816.553,E2 -23816.553} C_VEL
LIN {X 0,Y 159.287,Z 352.662,A -85,B 0,C 180,E1 -23819.514,E2 -23819.514} C_VEL
LIN {X 0,Y 155.811,Z 362.205,A -85,B 0,C 180,E1 -23823.193,E2 -23823.193} C_VEL
LIN {X 0,Y 152.861,Z 370.256,A -85,B 0,C 180,E1 -23827.093,E2 -23827.093} C_VEL
LIN {X 0,Y 150.785,Z 376.646,A -85,B 0,C 180,E1 -23830.962,E2 -23830.962} C_VEL
LIN {X 0,Y 149.126,Z 382.032,A -85,B 0,C 180,E1 -23834.981,E2 -23834.981} C_VEL
LIN {X 0,Y 148.16,Z 386.429,A -85,B 0,C 180,E1 -23839.066,E2 -23839.066} C_VEL
LIN {X 0,Y 147.695,Z 389.897,A -85,B 0,C 180,E1 -23843.172,E2 -23843.172} C_VEL
LIN {X 0,Y 147.649,Z 393.153,A -85,B 0,C 180,E1 -23848.614,E2 -23848.614} C_VEL
LIN {X 0,Y 147.627,Z 394.629,A -85,B 0,C 180,E1 -23852.733,E2 -23852.733} C_VEL
LIN {X 0,Y 147.843,Z 395.435,A -85,B 0,C 180,E1 -23858.203,E2 -23858.203} C_VEL
LIN {X 0,Y 148.985,Z 394.938,A -85,B 0,C 180,E1 -23863.646,E2 -23863.646} C_VEL
LIN {X 0,Y 151.32,Z 393.151,A -85,B 0,C 180,E1 -23868.976,E2 -23868.976} C_VEL
LIN {X 0,Y 154.924,Z 390.039,A -85,B 0,C 180,E1 -23874.101,E2 -23874.101} C_VEL
LIN {X 0,Y 159.574,Z 385.523,A -85,B 0,C 180,E1 -23878.981,E2 -23878.981} C_VEL
LIN {X 0,Y 163.865,Z 381.086,A -85,B 0,C 180,E1 -23882.423,E2 -23882.423} C_VEL
LIN {X 0,Y 169.627,Z 374.725,A -85,B 0,C 180,E1 -23886.19,E2 -23886.19} C_VEL
LIN {X 0,Y 176.159,Z 366.857,A -85,B 0,C 180,E1 -23889.671,E2 -23889.671} C_VEL
LIN {X 0,Y 182.278,Z 358.665,A -85,B 0,C 180,E1 -23892.438,E2 -23892.438} C_VEL
LIN {X 0,Y 187.822,Z 350.229,A -85,B 0,C 180,E1 -23894.726,E2 -23894.726} C_VEL
LIN {X 0,Y 194.461,Z 339.026,A -85,B 0,C 180,E1 -23897.046,E2 -23897.046} C_VEL
LIN {X 0,Y 200.425,Z 327.21,A -85,B 0,C 180,E1 -23898.934,E2 -23898.934} C_VEL
LIN {X 0,Y 205.405,Z 315.618,A -85,B 0,C 180,E1 -23900.344,E2 -23900.344} C_VEL
LIN {X 0,Y 210.218,Z 302.021,A -85,B 0,C 180,E1 -23901.592,E2 -23901.592} C_VEL
LIN {X 0,Y 214.073,Z 287.873,A -85,B 0,C 180,E1 -23902.515,E2 -23902.515} C_VEL
LIN {X 0,Y 216.755,Z 274.034,A -85,B 0,C 180,E1 -23903.146,E2 -23903.146} C_VEL
LIN {X 0,Y 218.501,Z 258.412,A -85,B 0,C 180,E1 -23903.637,E2 -23903.637} C_VEL
LIN {X 0,Y 220.891,Z 229.848,A -85,B 0,C 180,E1 -23904.433,E2 -23904.433} C_VEL
LIN {X 0,Y 216.996,Z 220.369,A -85,B 0,C 180,E1 -23907.047,E2 -23907.047} C_VEL
LIN {X 0,Y 213.245,Z 212.121,A -85,B 0,C 180,E1 -23909.877,E2 -23909.877} C_VEL
LIN {X 0,Y 209.714,Z 204.899,A -85,B 0,C 180,E1 -23912.975,E2 -23912.975} C_VEL
LIN {X 0,Y 207.676,Z 201.073,A -85,B 0,C 180,E1 -23915.013,E2 -23915.013} C_VEL
LIN {X 0,Y 205.063,Z 196.287,A -85,B 0,C 180,E1 -23918.072,E2 -23918.072} C_VEL
LIN {X 0,Y 202.418,Z 191.695,A -85,B 0,C 180,E1 -23922.156,E2 -23922.156} C_VEL
LIN {X 0,Y 199.839,Z 187.624,A -85,B 0,C 180,E1 -23930.122,E2 -23930.122} C_VEL
LIN {X 0,Y 199.808,Z 186.636,A -85,B 0,C 180,E1 -23931.906,E2 -23931.906} C_VEL
LIN {X 0,Y 199.886,Z 187.122,A -85,B 0,C 180,E1 -23934.206,E2 -23934.206} C_VEL
LIN {X 0,Y 200.605,Z 188.988,A -85,B 0,C 180,E1 -23937.986,E2 -23937.986} C_VEL
LIN {X 0,Y 202.823,Z 192.052,A -85,B 0,C 180,E1 -23942.94,E2 -23942.94} C_VEL
LIN {X 0,Y 205.027,Z 195.594,A -85,B 0,C 180,E1 -23946.218,E2 -23946.218} C_VEL
LIN {X 0,Y 208.548,Z 201.132,A -85,B 0,C 180,E1 -23950.141,E2 -23950.141} C_VEL
LIN {X 0,Y 211.159,Z 205.433,A -85,B 0,C 180,E1 -23952.548,E2 -23952.548} C_VEL
LIN {X 0,Y 214.843,Z 211.526,A -85,B 0,C 180,E1 -23955.474,E2 -23955.474} C_VEL
LIN {X 0,Y 218.815,Z 218.869,A -85,B 0,C 180,E1 -23958.213,E2 -23958.213} C_VEL
LIN {X 0,Y 221.371,Z 224.509,A -85,B 0,C 180,E1 -23959.854,E2 -23959.854} C_VEL
LIN {X 0,Y 217.803,Z 263.917,A -85,B 0,C 180,E1 -23960.937,E2 -23960.937} C_VEL
LIN {X 0,Y 215.324,Z 278.567,A -85,B 0,C 180,E1 -23961.583,E2 -23961.583} C_VEL
LIN {X 0,Y 211.988,Z 292.152,A -85,B 0,C 180,E1 -23962.455,E2 -23962.455} C_VEL
LIN {X 0,Y 208.023,Z 304.769,A -85,B 0,C 180,E1 -23963.587,E2 -23963.587} C_VEL
LIN {X 0,Y 203.236,Z 317.101,A -85,B 0,C 180,E1 -23965.043,E2 -23965.043} C_VEL
LIN {X 0,Y 197.792,Z 328.644,A -85,B 0,C 180,E1 -23966.774,E2 -23966.774} C_VEL
LIN {X 0,Y 191.693,Z 339.69,A -85,B 0,C 180,E1 -23968.911,E2 -23968.911} C_VEL
LIN {X 0,Y 185.357,Z 349.72,A -85,B 0,C 180,E1 -23971.443,E2 -23971.443} C_VEL
LIN {X 0,Y 178.808,Z 358.726,A -85,B 0,C 180,E1 -23974.366,E2 -23974.366} C_VEL
LIN {X 0,Y 172.613,Z 366.356,A -85,B 0,C 180,E1 -23977.631,E2 -23977.631} C_VEL
LIN {X 0,Y 167.367,Z 372.19,A -85,B 0,C 180,E1 -23980.896,E2 -23980.896} C_VEL
LIN {X 0,Y 162.51,Z 377.101,A -85,B 0,C 180,E1 -23984.469,E2 -23984.469} C_VEL
LIN {X 0,Y 158.316,Z 380.997,A -85,B 0,C 180,E1 -23988.245,E2 -23988.245} C_VEL
LIN {X 0,Y 153.78,Z 384.714,A -85,B 0,C 180,E1 -23993.546,E2 -23993.546} C_VEL
LIN {X 0,Y 150.481,Z 386.891,A -85,B 0,C 180,E1 -23999.083,E2 -23999.083} C_VEL
LIN {X 0,Y 148.417,Z 387.597,A -85,B 0,C 180,E1 -24004.771,E2 -24004.771} C_VEL
LIN {X 0,Y 147.399,Z 386.836,A -85,B 0,C 180,E1 -24010.499,E2 -24010.499} C_VEL
LIN {X 0,Y 147.257,Z 385.916,A -85,B 0,C 180,E1 -24013.356,E2 -24013.356} C_VEL
LIN {X 0,Y 147.419,Z 383.018,A -85,B 0,C 180,E1 -24019.003,E2 -24019.003} C_VEL
LIN {X 0,Y 148.342,Z 379.058,A -85,B 0,C 180,E1 -24024.114,E2 -24024.114} C_VEL
LIN {X 0,Y 149.634,Z 374.336,A -85,B 0,C 180,E1 -24028.651,E2 -24028.651} C_VEL
LIN {X 0,Y 151.656,Z 368.049,A -85,B 0,C 180,E1 -24033.317,E2 -24033.317} C_VEL
LIN {X 0,Y 154.593,Z 360.199,A -85,B 0,C 180,E1 -24037.835,E2 -24037.835} C_VEL
LIN {X 0,Y 158.013,Z 351.07,A -85,B 0,C 180,E1 -24041.952,E2 -24041.952} C_VEL
LIN {X 0,Y 161.157,Z 342.173,A -85,B 0,C 180,E1 -24045.165,E2 -24045.165} C_VEL
LIN {X 0,Y 164.461,Z 332.322,A -85,B 0,C 180,E1 -24048.044,E2 -24048.044} C_VEL
LIN {X 0,Y 167.934,Z 321.663,A -85,B 0,C 180,E1 -24050.514,E2 -24050.514} C_VEL
LIN {X 0,Y 171.189,Z 310.224,A -85,B 0,C 180,E1 -24052.633,E2 -24052.633} C_VEL
LIN {X 0,Y 174.204,Z 297.843,A -85,B 0,C 180,E1 -24054.422,E2 -24054.422} C_VEL
LIN {X 0,Y 176.761,Z 284.214,A -85,B 0,C 180,E1 -24055.932,E2 -24055.932} C_VEL
LIN {X 0,Y 178.733,Z 270.091,A -85,B 0,C 180,E1 -24057.039,E2 -24057.039} C_VEL
LIN {X 0,Y 180.031,Z 256.619,A -85,B 0,C 180,E1 -24057.693,E2 -24057.693} C_VEL
LIN {X 0,Y 184.12,Z 194.893,A -85,B 0,C 180,E1 -24059.786,E2 -24059.786} C_VEL
LIN {X 0,Y 182.391,Z 190.245,A -85,B 0,C 180,E1 -24060.474,E2 -24060.474} C_VEL
LIN {X 0,Y 177.272,Z 179.615,A -85,B 0,C 180,E1 -24062.455,E2 -24062.455} C_VEL
LIN {X 0,Y 171.184,Z 168.611,A -85,B 0,C 180,E1 -24064.949,E2 -24064.949} C_VEL
LIN {X 0,Y 165.413,Z 159.331,A -85,B 0,C 180,E1 -24067.523,E2 -24067.523} C_VEL
LIN {X 0,Y 159.846,Z 151.212,A -85,B 0,C 180,E1 -24070.261,E2 -24070.261} C_VEL
LIN {X 0,Y 157.001,Z 147.249,A -85,B 0,C 180,E1 -24071.787,E2 -24071.787} C_VEL
LIN {X 0,Y 154.581,Z 144.195,A -85,B 0,C 180,E1 -24073.144,E2 -24073.144} C_VEL
LIN {X 0,Y 153.612,Z 142.541,A -85,B 0,C 180,E1 -24073.741,E2 -24073.741} C_VEL
LIN {X 0,Y 151.409,Z 140.485,A -85,B 0,C 180,E1 -24075.023,E2 -24075.023} C_VEL
LIN {X 0,Y 150.337,Z 137.963,A -85,B 0,C 180,E1 -24075.8,E2 -24075.8} C_VEL
LIN {X 0,Y 150.25,Z 137.377,A -85,B 0,C 180,E1 -24075.974,E2 -24075.974} C_VEL
LIN {X 0,Y 150.213,Z 137.38,A -85,B 0,C 180,E1 -24079.093,E2 -24079.093} C_VEL
LIN {X 0,Y 150.215,Z 137.36,A -85,B 0,C 180,E1 -24082.683,E2 -24082.683} C_VEL
LIN {X 0,Y 150.195,Z 137.395,A -85,B 0,C 180,E1 -24087.372,E2 -24087.372} C_VEL
LIN {X 0,Y 150.225,Z 137.355,A -85,B 0,C 180,E1 -24092.724,E2 -24092.724} C_VEL
LIN {X 0,Y 150.372,Z 137.369,A -85,B 0,C 180,E1 -24099.176,E2 -24099.176} C_VEL
LIN {X 0,Y 150.382,Z 137.372,A -85,B 0,C 180,E1 -24103.725,E2 -24103.725} C_VEL
LIN {X 0,Y 150.674,Z 137.335,A -85,B 0,C 180,E1 -24109.256,E2 -24109.256} C_VEL
LIN {X 0,Y 150.748,Z 137.292,A -85,B 0,C 180,E1 -24111.969,E2 -24111.969} C_VEL
LIN {X 0,Y 151.21,Z 137.271,A -85,B 0,C 180,E1 -24120.009,E2 -24120.009} C_VEL
LIN {X 0,Y 150.738,Z 137.321,A -85,B 0,C 180,E1 -24128.049,E2 -24128.049} C_VEL
LIN {X 0,Y 150.609,Z 137.342,A -85,B 0,C 180,E1 -24131.516,E2 -24131.516} C_VEL
LIN {X 0,Y 150.378,Z 137.372,A -85,B 0,C 180,E1 -24136.293,E2 -24136.293} C_VEL
LIN {X 0,Y 150.349,Z 137.379,A -85,B 0,C 180,E1 -24140.801,E2 -24140.801} C_VEL
LIN {X 0,Y 150.242,Z 137.379,A -85,B 0,C 180,E1 -24147.46,E2 -24147.46} C_VEL
LIN {X 0,Y 150.237,Z 137.471,A -85,B 0,C 180,E1 -24147.735,E2 -24147.735} C_VEL
LIN {X 0,Y 151.071,Z 140.001,A -85,B 0,C 180,E1 -24148.393,E2 -24148.393} C_VEL
LIN {X 0,Y 153.047,Z 142.213,A -85,B 0,C 180,E1 -24149.589,E2 -24149.589} C_VEL
LIN {X 0,Y 154.115,Z 143.128,A -85,B 0,C 180,E1 -24150.187,E2 -24150.187} C_VEL
LIN {X 0,Y 155.933,Z 146.168,A -85,B 0,C 180,E1 -24151.28,E2 -24151.28} C_VEL
LIN {X 0,Y 157.726,Z 148.199,A -85,B 0,C 180,E1 -24152.239,E2 -24152.239} C_VEL
LIN {X 0,Y 161.915,Z 154.289,A -85,B 0,C 180,E1 -24154.418,E2 -24154.418} C_VEL
LIN {X 0,Y 166.797,Z 161.553,A -85,B 0,C 180,E1 -24156.738,E2 -24156.738} C_VEL
LIN {X 0,Y 170.002,Z 167.123,A -85,B 0,C 180,E1 -24158.189,E2 -24158.189} C_VEL
LIN {X 0,Y 175.768,Z 179.62,A -85,B 0,C 180,E1 -24160.731,E2 -24160.731} C_VEL
LIN {X 0,Y 180.106,Z 190.708,A -85,B 0,C 180,E1 -24162.565,E2 -24162.565} C_VEL
LIN {X 0,Y 183.743,Z 201.199,A -85,B 0,C 180,E1 -24164.063,E2 -24164.063} C_VEL
LIN {X 0,Y 179.432,Z 270.379,A -85,B 0,C 180,E1 -24166.541,E2 -24166.541} C_VEL
LIN {X 0,Y 177.619,Z 285.117,A -85,B 0,C 180,E1 -24167.445,E2 -24167.445} C_VEL
LIN {X 0,Y 175.049,Z 299.162,A -85,B 0,C 180,E1 -24168.709,E2 -24168.709} C_VEL
LIN {X 0,Y 172.068,Z 312.254,A -85,B 0,C 180,E1 -24170.347,E2 -24170.347} C_VEL
LIN {X 0,Y 168.661,Z 324.549,A -85,B 0,C 180,E1 -24172.356,E2 -24172.356} C_VEL
LIN {X 0,Y 165.814,Z 334.15,A -85,B 0,C 180,E1 -24174.357,E2 -24174.357} C_VEL
LIN {X 0,Y 163.452,Z 340.99,A -85,B 0,C 180,E1 -24176.02,E2 -24176.02} C_VEL
LIN {X 0,Y 162.796,Z 342.999,A -85,B 0,C 180,E1 -24176.553,E2 -24176.553} C_VEL
LIN {X 0,Y 160.69,Z 347.436,A -85,B 0,C 180,E1 -24177.716,E2 -24177.716} C_VEL
LIN {X 0,Y 155.518,Z 354.222,A -85,B 0,C 180,E1 -24179.553,E2 -24179.553} C_VEL
LIN {X 0,Y 150.356,Z 360.539,A -85,B 0,C 180,E1 -24181.683,E2 -24181.683} C_VEL
LIN {X 0,Y 148.324,Z 364.199,A -85,B 0,C 180,E1 -24183.279,E2 -24183.279} C_VEL
LIN {X 0,Y 145.48,Z 371.68,A -85,B 0,C 180,E1 -24187.269,E2 -24187.269} C_VEL
LIN {X 0,Y 143.375,Z 377.942,A -85,B 0,C 180,E1 -24191.425,E2 -24191.425} C_VEL
LIN {X 0,Y 141.788,Z 383.097,A -85,B 0,C 180,E1 -24195.655,E2 -24195.655} C_VEL
LIN {X 0,Y 140.777,Z 388.386,A -85,B 0,C 180,E1 -24201.391,E2 -24201.391} C_VEL
LIN {X 0,Y 140.522,Z 392.095,A -85,B 0,C 180,E1 -24207.137,E2 -24207.137} C_VEL
LIN {X 0,Y 140.588,Z 393.663,A -85,B 0,C 180,E1 -24210.691,E2 -24210.691} C_VEL
LIN {X 0,Y 140.563,Z 394.946,A -85,B 0,C 180,E1 -24215.743,E2 -24215.743} C_VEL
LIN {X 0,Y 141.31,Z 395.169,A -85,B 0,C 180,E1 -24221.479,E2 -24221.479} C_VEL
LIN {X 0,Y 143.105,Z 394.102,A -85,B 0,C 180,E1 -24227.141,E2 -24227.141} C_VEL
LIN {X 0,Y 146.34,Z 391.74,A -85,B 0,C 180,E1 -24232.598,E2 -24232.598} C_VEL
LIN {X 0,Y 150.736,Z 388.022,A -85,B 0,C 180,E1 -24237.795,E2 -24237.795} C_VEL
LIN {X 0,Y 156.307,Z 382.845,A -85,B 0,C 180,E1 -24242.657,E2 -24242.657} C_VEL
LIN {X 0,Y 161.251,Z 377.865,A -85,B 0,C 180,E1 -24246.047,E2 -24246.047} C_VEL
LIN {X 0,Y 167.733,Z 370.778,A -85,B 0,C 180,E1 -24249.72,E2 -24249.72} C_VEL
LIN {X 0,Y 174.979,Z 362.045,A -85,B 0,C 180,E1 -24253.067,E2 -24253.067} C_VEL
LIN {X 0,Y 181.647,Z 352.677,A -85,B 0,C 180,E1 -24255.851,E2 -24255.851} C_VEL
LIN {X 0,Y 188.534,Z 341.956,A -85,B 0,C 180,E1 -24258.21,E2 -24258.21} C_VEL
LIN {X 0,Y 194.648,Z 330.782,A -85,B 0,C 180,E1 -24260.112,E2 -24260.112} C_VEL
LIN {X 0,Y 200.359,Z 318.475,A -85,B 0,C 180,E1 -24261.711,E2 -24261.711} C_VEL
LIN {X 0,Y 204.94,Z 306.646,A -85,B 0,C 180,E1 -24262.878,E2 -24262.878} C_VEL
LIN {X 0,Y 208.984,Z 293.744,A -85,B 0,C 180,E1 -24263.818,E2 -24263.818} C_VEL
LIN {X 0,Y 212.135,Z 280.502,A -85,B 0,C 180,E1 -24264.508,E2 -24264.508} C_VEL
LIN {X 0,Y 214.303,Z 265.982,A -85,B 0,C 180,E1 -24265.075,E2 -24265.075} C_VEL
LIN {X 0,Y 217.278,Z 233.024,A -85,B 0,C 180,E1 -24265.975,E2 -24265.975} C_VEL
LIN {X 0,Y 213.936,Z 224.705,A -85,B 0,C 180,E1 -24268.406,E2 -24268.406} C_VEL
LIN {X 0,Y 210.605,Z 216.971,A -85,B 0,C 180,E1 -24271.177,E2 -24271.177} C_VEL
LIN {X 0,Y 207.632,Z 210.653,A -85,B 0,C 180,E1 -24273.999,E2 -24273.999} C_VEL
LIN {X 0,Y 206,Z 207.434,A -85,B 0,C 180,E1 -24275.748,E2 -24275.748} C_VEL
LIN {X 0,Y 203.52,Z 202.66,A -85,B 0,C 180,E1 -24278.852,E2 -24278.852} C_VEL
LIN {X 0,Y 201.072,Z 198.429,A -85,B 0,C 180,E1 -24282.95,E2 -24282.95} C_VEL
LIN {X 0,Y 198.91,Z 194.245,A -85,B 0,C 180,E1 -24290.965,E2 -24290.965} C_VEL
LIN {X 0,Y 198.924,Z 193.683,A -85,B 0,C 180,E1 -24291.869,E2 -24291.869} C_VEL
LIN {X 0,Y 198.996,Z 194.179,A -85,B 0,C 180,E1 -24294.18,E2 -24294.18} C_VEL
LIN {X 0,Y 199.705,Z 196.1,A -85,B 0,C 180,E1 -24297.977,E2 -24297.977} C_VEL
LIN {X 0,Y 201.661,Z 198.942,A -85,B 0,C 180,E1 -24302.52,E2 -24302.52} C_VEL
LIN {X 0,Y 203.754,Z 202.399,A -85,B 0,C 180,E1 -24305.795,E2 -24305.795} C_VEL
LIN {X 0,Y 206.926,Z 207.677,A -85,B 0,C 180,E1 -24309.511,E2 -24309.511} C_VEL
LIN {X 0,Y 209.409,Z 211.935,A -85,B 0,C 180,E1 -24311.917,E2 -24311.917} C_VEL
LIN {X 0,Y 212.817,Z 217.808,A -85,B 0,C 180,E1 -24314.761,E2 -24314.761} C_VEL
LIN {X 0,Y 216.3,Z 224.572,A -85,B 0,C 180,E1 -24317.318,E2 -24317.318} C_VEL
LIN {X 0,Y 217.7,Z 227.801,A -85,B 0,C 180,E1 -24318.286,E2 -24318.286} C_VEL
LIN {X 0,Y 214.216,Z 264.881,A -85,B 0,C 180,E1 -24319.325,E2 -24319.325} C_VEL
LIN {X 0,Y 211.687,Z 279.225,A -85,B 0,C 180,E1 -24319.963,E2 -24319.963} C_VEL
LIN {X 0,Y 208.532,Z 291.638,A -85,B 0,C 180,E1 -24320.727,E2 -24320.727} C_VEL
LIN {X 0,Y 204.457,Z 304.421,A -85,B 0,C 180,E1 -24321.853,E2 -24321.853} C_VEL
LIN {X 0,Y 199.13,Z 317.738,A -85,B 0,C 180,E1 -24323.411,E2 -24323.411} C_VEL
LIN {X 0,Y 193.265,Z 329.671,A -85,B 0,C 180,E1 -24325.208,E2 -24325.208} C_VEL
LIN {X 0,Y 186.941,Z 340.61,A -85,B 0,C 180,E1 -24327.349,E2 -24327.349} C_VEL
LIN {X 0,Y 180.373,Z 350.512,A -85,B 0,C 180,E1 -24329.889,E2 -24329.889} C_VEL
LIN {X 0,Y 173.559,Z 359.39,A -85,B 0,C 180,E1 -24332.829,E2 -24332.829} C_VEL
LIN {X 0,Y 167.315,Z 366.687,A -85,B 0,C 180,E1 -24336.009,E2 -24336.009} C_VEL
LIN {X 0,Y 160.697,Z 373.589,A -85,B 0,C 180,E1 -24340.057,E2 -24340.057} C_VEL
LIN {X 0,Y 155.674,Z 378.293,A -85,B 0,C 180,E1 -24343.748,E2 -24343.748} C_VEL
LIN {X 0,Y 150.886,Z 382.341,A -85,B 0,C 180,E1 -24348.165,E2 -24348.165} C_VEL
LIN {X 0,Y 147.75,Z 384.671,A -85,B 0,C 180,E1 -24351.798,E2 -24351.798} C_VEL
LIN {X 0,Y 144.038,Z 386.959,A -85,B 0,C 180,E1 -24357.535,E2 -24357.535} C_VEL
LIN {X 0,Y 141.645,Z 387.776,A -85,B 0,C 180,E1 -24363.473,E2 -24363.473} C_VEL
LIN {X 0,Y 140.387,Z 387.16,A -85,B 0,C 180,E1 -24369.482,E2 -24369.482} C_VEL
LIN {X 0,Y 140.178,Z 386.311,A -85,B 0,C 180,E1 -24372.489,E2 -24372.489} C_VEL
LIN {X 0,Y 140.118,Z 385.099,A -85,B 0,C 180,E1 -24375.472,E2 -24375.472} C_VEL
LIN {X 0,Y 140.688,Z 381.582,A -85,B 0,C 180,E1 -24381.377,E2 -24381.377} C_VEL
LIN {X 0,Y 141.633,Z 377.992,A -85,B 0,C 180,E1 -24385.727,E2 -24385.727} C_VEL
LIN {X 0,Y 142.961,Z 373.442,A -85,B 0,C 180,E1 -24389.996,E2 -24389.996} C_VEL
LIN {X 0,Y 145.315,Z 366.88,A -85,B 0,C 180,E1 -24394.851,E2 -24394.851} C_VEL
LIN {X 0,Y 148.49,Z 358.741,A -85,B 0,C 180,E1 -24399.531,E2 -24399.531} C_VEL
LIN {X 0,Y 151.856,Z 350.216,A -85,B 0,C 180,E1 -24403.376,E2 -24403.376} C_VEL
LIN {X 0,Y 154.934,Z 341.78,A -85,B 0,C 180,E1 -24406.466,E2 -24406.466} C_VEL
LIN {X 0,Y 158.099,Z 332.875,A -85,B 0,C 180,E1 -24409.134,E2 -24409.134} C_VEL
LIN {X 0,Y 161.697,Z 322.294,A -85,B 0,C 180,E1 -24411.677,E2 -24411.677} C_VEL
LIN {X 0,Y 165.548,Z 309.352,A -85,B 0,C 180,E1 -24414.114,E2 -24414.114} C_VEL
LIN {X 0,Y 168.863,Z 295.73,A -85,B 0,C 180,E1 -24416.075,E2 -24416.075} C_VEL
LIN {X 0,Y 171.334,Z 282.671,A -85,B 0,C 180,E1 -24417.478,E2 -24417.478} C_VEL
LIN {X 0,Y 173.263,Z 268.674,A -85,B 0,C 180,E1 -24418.543,E2 -24418.543} C_VEL
LIN {X 0,Y 174.648,Z 253.794,A -85,B 0,C 180,E1 -24419.21,E2 -24419.21} C_VEL
LIN {X 0,Y 178.526,Z 196.37,A -85,B 0,C 180,E1 -24421.201,E2 -24421.201} C_VEL
LIN {X 0,Y 173.66,Z 185.677,A -85,B 0,C 180,E1 -24423.19,E2 -24423.19} C_VEL
LIN {X 0,Y 167.451,Z 174.03,A -85,B 0,C 180,E1 -24425.879,E2 -24425.879} C_VEL
LIN {X 0,Y 161.402,Z 164.096,A -85,B 0,C 180,E1 -24428.749,E2 -24428.749} C_VEL
LIN {X 0,Y 156.292,Z 156.503,A -85,B 0,C 180,E1 -24431.433,E2 -24431.433} C_VEL
LIN {X 0,Y 153.741,Z 152.93,A -85,B 0,C 180,E1 -24432.883,E2 -24432.883} C_VEL
LIN {X 0,Y 151.142,Z 149.338,A -85,B 0,C 180,E1 -24434.449,E2 -24434.449} C_VEL
LIN {X 0,Y 149.668,Z 147.686,A -85,B 0,C 180,E1 -24435.355,E2 -24435.355} C_VEL
LIN {X 0,Y 147.635,Z 144.821,A -85,B 0,C 180,E1 -24436.716,E2 -24436.716} C_VEL
LIN {X 0,Y 147.11,Z 143.766,A -85,B 0,C 180,E1 -24437.11,E2 -24437.11} C_VEL
LIN {X 0,Y 144.647,Z 141.795,A -85,B 0,C 180,E1 -24438.772,E2 -24438.772} C_VEL
LIN {X 0,Y 143.355,Z 139.317,A -85,B 0,C 180,E1 -24439.839,E2 -24439.839} C_VEL
LIN {X 0,Y 143.108,Z 138.249,A -85,B 0,C 180,E1 -24440.173,E2 -24440.173} C_VEL
LIN {X 0,Y 143.146,Z 138.277,A -85,B 0,C 180,E1 -24446.571,E2 -24446.571} C_VEL
LIN {X 0,Y 143.17,Z 138.229,A -85,B 0,C 180,E1 -24452.07,E2 -24452.07} C_VEL
LIN {X 0,Y 143.293,Z 138.252,A -85,B 0,C 180,E1 -24458.718,E2 -24458.718} C_VEL
LIN {X 0,Y 143.32,Z 138.257,A -85,B 0,C 180,E1 -24462.899,E2 -24462.899} C_VEL
LIN {X 0,Y 143.588,Z 138.222,A -85,B 0,C 180,E1 -24468.719,E2 -24468.719} C_VEL
LIN {X 0,Y 143.669,Z 138.176,A -85,B 0,C 180,E1 -24471.571,E2 -24471.571} C_VEL
LIN {X 0,Y 144.168,Z 138.148,A -85,B 0,C 180,E1 -24480.009,E2 -24480.009} C_VEL
LIN {X 0,Y 143.659,Z 138.206,A -85,B 0,C 180,E1 -24488.448,E2 -24488.448} C_VEL
LIN {X 0,Y 143.543,Z 138.221,A -85,B 0,C 180,E1 -24491.722,E2 -24491.722} C_VEL
LIN {X 0,Y 143.313,Z 138.249,A -85,B 0,C 180,E1 -24497.121,E2 -24497.121} C_VEL
LIN {X 0,Y 143.275,Z 138.26,A -85,B 0,C 180,E1 -24501.264,E2 -24501.264} C_VEL
LIN {X 0,Y 143.165,Z 138.273,A -85,B 0,C 180,E1 -24503.516,E2 -24503.516} C_VEL
LIN {X 0,Y 144.064,Z 140.956,A -85,B 0,C 180,E1 -24504.411,E2 -24504.411} C_VEL
LIN {X 0,Y 146.267,Z 143.299,A -85,B 0,C 180,E1 -24505.981,E2 -24505.981} C_VEL
LIN {X 0,Y 147.298,Z 144.141,A -85,B 0,C 180,E1 -24506.656,E2 -24506.656} C_VEL
LIN {X 0,Y 149.348,Z 147.426,A -85,B 0,C 180,E1 -24508.081,E2 -24508.081} C_VEL
LIN {X 0,Y 151.206,Z 149.365,A -85,B 0,C 180,E1 -24509.221,E2 -24509.221} C_VEL
LIN {X 0,Y 153.756,Z 152.947,A -85,B 0,C 180,E1 -24510.764,E2 -24510.764} C_VEL
LIN {X 0,Y 158.238,Z 159.418,A -85,B 0,C 180,E1 -24513.255,E2 -24513.255} C_VEL
LIN {X 0,Y 164.479,Z 169.07,A -85,B 0,C 180,E1 -24516.369,E2 -24516.369} C_VEL
LIN {X 0,Y 169.701,Z 180.156,A -85,B 0,C 180,E1 -24518.863,E2 -24518.863} C_VEL
LIN {X 0,Y 174.664,Z 192.717,A -85,B 0,C 180,E1 -24521.128,E2 -24521.128} C_VEL
LIN {X 0,Y 178.147,Z 202.985,A -85,B 0,C 180,E1 -24522.675,E2 -24522.675} C_VEL
LIN {X 0,Y 173.774,Z 270.624,A -85,B 0,C 180,E1 -24525.157,E2 -24525.157} C_VEL
LIN {X 0,Y 171.894,Z 285.213,A -85,B 0,C 180,E1 -24526.075,E2 -24526.075} C_VEL
LIN {X 0,Y 169.231,Z 299.183,A -85,B 0,C 180,E1 -24527.361,E2 -24527.361} C_VEL
LIN {X 0,Y 166.141,Z 312.23,A -85,B 0,C 180,E1 -24529.034,E2 -24529.034} C_VEL
LIN {X 0,Y 162.597,Z 324.5,A -85,B 0,C 180,E1 -24531.09,E2 -24531.09} C_VEL
LIN {X 0,Y 159.625,Z 334.069,A -85,B 0,C 180,E1 -24533.143,E2 -24533.143} C_VEL
LIN {X 0,Y 157.155,Z 340.898,A -85,B 0,C 180,E1 -24534.851,E2 -24534.851} C_VEL
LIN {X 0,Y 153.132,Z 351.645,A -85,B 0,C 180,E1 -24538.148,E2 -24538.148} C_VEL
LIN {X 0,Y 149.437,Z 361.338,A -85,B 0,C 180,E1 -24541.951,E2 -24541.951} C_VEL
LIN {X 0,Y 148.324,Z 364.199,A -85,B 0,C 180,E1 -24543.279,E2 -24543.279} C_VEL
LIN {X 0,Y 146.394,Z 367.719,A -85,B 0,C 180,E1 -24544.969,E2 -24544.969} C_VEL
LIN {X 0,Y 141.67,Z 372.98,A -85,B 0,C 180,E1 -24547.737,E2 -24547.737} C_VEL
LIN {X 0,Y 137.134,Z 377.718,A -85,B 0,C 180,E1 -24550.816,E2 -24550.816} C_VEL
LIN {X 0,Y 135.559,Z 380.344,A -85,B 0,C 180,E1 -24552.94,E2 -24552.94} C_VEL
LIN {X 0,Y 134.171,Z 385.462,A -85,B 0,C 180,E1 -24557.91,E2 -24557.91} C_VEL
LIN {X 0,Y 133.588,Z 389.02,A -85,B 0,C 180,E1 -24562.447,E2 -24562.447} C_VEL
LIN {X 0,Y 133.424,Z 391.733,A -85,B 0,C 180,E1 -24566.985,E2 -24566.985} C_VEL
LIN {X 0,Y 133.55,Z 393.076,A -85,B 0,C 180,E1 -24570.004,E2 -24570.004} C_VEL
LIN {X 0,Y 133.475,Z 394.055,A -85,B 0,C 180,E1 -24573.023,E2 -24573.023} C_VEL
LIN {X 0,Y 133.756,Z 395.004,A -85,B 0,C 180,E1 -24579.074,E2 -24579.074} C_VEL
LIN {X 0,Y 135.149,Z 394.656,A -85,B 0,C 180,E1 -24585.075,E2 -24585.075} C_VEL
LIN {X 0,Y 137.905,Z 393.024,A -85,B 0,C 180,E1 -24590.904,E2 -24590.904} C_VEL
LIN {X 0,Y 141.997,Z 390.073,A -85,B 0,C 180,E1 -24596.456,E2 -24596.456} C_VEL
LIN {X 0,Y 147.262,Z 385.725,A -85,B 0,C 180,E1 -24601.67,E2 -24601.67} C_VEL
LIN {X 0,Y 153.763,Z 379.855,A -85,B 0,C 180,E1 -24606.459,E2 -24606.459} C_VEL
LIN {X 0,Y 160.321,Z 373.289,A -85,B 0,C 180,E1 -24610.29,E2 -24610.29} C_VEL
LIN {X 0,Y 167.68,Z 365.176,A -85,B 0,C 180,E1 -24613.759,E2 -24613.759} C_VEL
LIN {X 0,Y 174.936,Z 355.884,A -85,B 0,C 180,E1 -24616.773,E2 -24616.773} C_VEL
LIN {X 0,Y 181.436,Z 346.576,A -85,B 0,C 180,E1 -24619.06,E2 -24619.06} C_VEL
LIN {X 0,Y 188.32,Z 335.233,A -85,B 0,C 180,E1 -24621.177,E2 -24621.177} C_VEL
LIN {X 0,Y 194.073,Z 324.008,A -85,B 0,C 180,E1 -24622.82,E2 -24622.82} C_VEL
LIN {X 0,Y 199.44,Z 311.739,A -85,B 0,C 180,E1 -24624.148,E2 -24624.148} C_VEL
LIN {X 0,Y 203.891,Z 299.215,A -85,B 0,C 180,E1 -24625.169,E2 -24625.169} C_VEL
LIN {X 0,Y 207.676,Z 285.36,A -85,B 0,C 180,E1 -24625.998,E2 -24625.998} C_VEL
LIN {X 0,Y 210.318,Z 271.415,A -85,B 0,C 180,E1 -24626.59,E2 -24626.59} C_VEL
LIN {X 0,Y 212.71,Z 248.447,A -85,B 0,C 180,E1 -24627.241,E2 -24627.241} C_VEL
LIN {X 0,Y 213.772,Z 236.2,A -85,B 0,C 180,E1 -24627.598,E2 -24627.598} C_VEL
LIN {X 0,Y 210.778,Z 228.323,A -85,B 0,C 180,E1 -24630.042,E2 -24630.042} C_VEL
LIN {X 0,Y 207.715,Z 221.065,A -85,B 0,C 180,E1 -24632.855,E2 -24632.855} C_VEL
LIN {X 0,Y 204.995,Z 214.961,A -85,B 0,C 180,E1 -24635.763,E2 -24635.763} C_VEL
LIN {X 0,Y 202.112,Z 209.267,A -85,B 0,C 180,E1 -24639.492,E2 -24639.492} C_VEL
LIN {X 0,Y 199.947,Z 205.292,A -85,B 0,C 180,E1 -24643.392,E2 -24643.392} C_VEL
LIN {X 0,Y 198.017,Z 201.018,A -85,B 0,C 180,E1 -24651.567,E2 -24651.567} C_VEL
LIN {X 0,Y 198.084,Z 201.153,A -85,B 0,C 180,E1 -24653.883,E2 -24653.883} C_VEL
LIN {X 0,Y 198.615,Z 202.803,A -85,B 0,C 180,E1 -24657.267,E2 -24657.267} C_VEL
LIN {X 0,Y 200.522,Z 205.856,A -85,B 0,C 180,E1 -24662.118,E2 -24662.118} C_VEL
LIN {X 0,Y 202.818,Z 209.933,A -85,B 0,C 180,E1 -24665.839,E2 -24665.839} C_VEL
LIN {X 0,Y 205.538,Z 214.591,A -85,B 0,C 180,E1 -24669.099,E2 -24669.099} C_VEL
LIN {X 0,Y 208.804,Z 220.285,A -85,B 0,C 180,E1 -24672.291,E2 -24672.291} C_VEL
LIN {X 0,Y 212.823,Z 228.053,A -85,B 0,C 180,E1 -24675.625,E2 -24675.625} C_VEL
LIN {X 0,Y 214.237,Z 231.237,A -85,B 0,C 180,E1 -24676.7,E2 -24676.7} C_VEL
LIN {X 0,Y 210.954,Z 264.89,A -85,B 0,C 180,E1 -24677.628,E2 -24677.628} C_VEL
LIN {X 0,Y 208.352,Z 279.296,A -85,B 0,C 180,E1 -24678.253,E2 -24678.253} C_VEL
LIN {X 0,Y 204.932,Z 292.327,A -85,B 0,C 180,E1 -24679.042,E2 -24679.042} C_VEL
LIN {X 0,Y 200.318,Z 306.118,A -85,B 0,C 180,E1 -24680.264,E2 -24680.264} C_VEL
LIN {X 0,Y 194.9,Z 318.991,A -85,B 0,C 180,E1 -24681.786,E2 -24681.786} C_VEL
LIN {X 0,Y 188.835,Z 330.776,A -85,B 0,C 180,E1 -24683.576,E2 -24683.576} C_VEL
LIN {X 0,Y 182.975,Z 340.506,A -85,B 0,C 180,E1 -24685.488,E2 -24685.488} C_VEL
LIN {X 0,Y 176.719,Z 349.602,A -85,B 0,C 180,E1 -24687.759,E2 -24687.759} C_VEL
LIN {X 0,Y 169.568,Z 358.696,A -85,B 0,C 180,E1 -24690.676,E2 -24690.676} C_VEL
LIN {X 0,Y 162.148,Z 367.023,A -85,B 0,C 180,E1 -24694.284,E2 -24694.284} C_VEL
LIN {X 0,Y 155.905,Z 373.234,A -85,B 0,C 180,E1 -24697.914,E2 -24697.914} C_VEL
LIN {X 0,Y 150.545,Z 378.015,A -85,B 0,C 180,E1 -24701.669,E2 -24701.669} C_VEL
LIN {X 0,Y 144.717,Z 382.638,A -85,B 0,C 180,E1 -24706.742,E2 -24706.742} C_VEL
LIN {X 0,Y 141.836,Z 384.628,A -85,B 0,C 180,E1 -24709.893,E2 -24709.893} C_VEL
LIN {X 0,Y 137.717,Z 387.028,A -85,B 0,C 180,E1 -24715.846,E2 -24715.846} C_VEL
LIN {X 0,Y 134.835,Z 387.969,A -85,B 0,C 180,E1 -24722.361,E2 -24722.361} C_VEL
LIN {X 0,Y 133.433,Z 387.446,A -85,B 0,C 180,E1 -24728.36,E2 -24728.36} C_VEL
LIN {X 0,Y 133.107,Z 386.573,A -85,B 0,C 180,E1 -24731.839,E2 -24731.839} C_VEL
LIN {X 0,Y 133.098,Z 384.021,A -85,B 0,C 180,E1 -24737.802,E2 -24737.802} C_VEL
LIN {X 0,Y 133.755,Z 381.04,A -85,B 0,C 180,E1 -24742.448,E2 -24742.448} C_VEL
LIN {X 0,Y 134.839,Z 377.227,A -85,B 0,C 180,E1 -24747.008,E2 -24747.008} C_VEL
LIN {X 0,Y 136.373,Z 372.515,A -85,B 0,C 180,E1 -24751.472,E2 -24751.472} C_VEL
LIN {X 0,Y 139.014,Z 365.65,A -85,B 0,C 180,E1 -24756.527,E2 -24756.527} C_VEL
LIN {X 0,Y 142.559,Z 357.119,A -85,B 0,C 180,E1 -24761.369,E2 -24761.369} C_VEL
LIN {X 0,Y 146.37,Z 347.867,A -85,B 0,C 180,E1 -24765.464,E2 -24765.464} C_VEL
LIN {X 0,Y 150.185,Z 337.509,A -85,B 0,C 180,E1 -24769.117,E2 -24769.117} C_VEL
LIN {X 0,Y 154.346,Z 326.562,A -85,B 0,C 180,E1 -24772.061,E2 -24772.061} C_VEL
LIN {X 0,Y 158.162,Z 314.64,A -85,B 0,C 180,E1 -24774.615,E2 -24774.615} C_VEL
LIN {X 0,Y 161.833,Z 301.435,A -85,B 0,C 180,E1 -24776.775,E2 -24776.775} C_VEL
LIN {X 0,Y 164.863,Z 287.481,A -85,B 0,C 180,E1 -24778.48,E2 -24778.48} C_VEL
LIN {X 0,Y 167.103,Z 273.605,A -85,B 0,C 180,E1 -24779.698,E2 -24779.698} C_VEL
LIN {X 0,Y 168.721,Z 260.039,A -85,B 0,C 180,E1 -24780.448,E2 -24780.448} C_VEL
LIN {X 0,Y 172.996,Z 198.393,A -85,B 0,C 180,E1 -24782.677,E2 -24782.677} C_VEL
LIN {X 0,Y 168.055,Z 187.755,A -85,B 0,C 180,E1 -24784.847,E2 -24784.847} C_VEL
LIN {X 0,Y 163.03,Z 178.229,A -85,B 0,C 180,E1 -24787.2,E2 -24787.2} C_VEL
LIN {X 0,Y 157.62,Z 169.135,A -85,B 0,C 180,E1 -24789.952,E2 -24789.952} C_VEL
LIN {X 0,Y 152.745,Z 161.695,A -85,B 0,C 180,E1 -24792.692,E2 -24792.692} C_VEL
LIN {X 0,Y 150.08,Z 157.979,A -85,B 0,C 180,E1 -24794.303,E2 -24794.303} C_VEL
LIN {X 0,Y 147.288,Z 154.084,A -85,B 0,C 180,E1 -24796.117,E2 -24796.117} C_VEL
LIN {X 0,Y 144.804,Z 150.738,A -85,B 0,C 180,E1 -24797.853,E2 -24797.853} C_VEL
LIN {X 0,Y 143.978,Z 149.729,A -85,B 0,C 180,E1 -24798.453,E2 -24798.453} C_VEL
LIN {X 0,Y 141.47,Z 146.93,A -85,B 0,C 180,E1 -24800.357,E2 -24800.357} C_VEL
LIN {X 0,Y 140.397,Z 144.783,A -85,B 0,C 180,E1 -24801.323,E2 -24801.323} C_VEL
LIN {X 0,Y 137.745,Z 142.925,A -85,B 0,C 180,E1 -24803.521,E2 -24803.521} C_VEL
LIN {X 0,Y 136.299,Z 140.341,A -85,B 0,C 180,E1 -24805.009,E2 -24805.009} C_VEL
LIN {X 0,Y 136.06,Z 139.151,A -85,B 0,C 180,E1 -24805.389,E2 -24805.389} C_VEL
LIN {X 0,Y 136.127,Z 139.105,A -85,B 0,C 180,E1 -24812.324,E2 -24812.324} C_VEL
LIN {X 0,Y 136.26,Z 139.127,A -85,B 0,C 180,E1 -24818.847,E2 -24818.847} C_VEL
LIN {X 0,Y 136.279,Z 139.121,A -85,B 0,C 180,E1 -24825.068,E2 -24825.068} C_VEL
LIN {X 0,Y 136.488,Z 139.107,A -85,B 0,C 180,E1 -24828.124,E2 -24828.124} C_VEL
LIN {X 0,Y 136.593,Z 139.06,A -85,B 0,C 180,E1 -24831.131,E2 -24831.131} C_VEL
LIN {X 0,Y 137.125,Z 139.026,A -85,B 0,C 180,E1 -24840.01,E2 -24840.01} C_VEL
LIN {X 0,Y 136.586,Z 139.091,A -85,B 0,C 180,E1 -24848.889,E2 -24848.889} C_VEL
LIN {X 0,Y 136.486,Z 139.099,A -85,B 0,C 180,E1 -24851.964,E2 -24851.964} C_VEL
LIN {X 0,Y 136.229,Z 139.184,A -85,B 0,C 180,E1 -24858.43,E2 -24858.43} C_VEL
LIN {X 0,Y 136.94,Z 141.459,A -85,B 0,C 180,E1 -24859.302,E2 -24859.302} C_VEL
LIN {X 0,Y 138.958,Z 143.872,A -85,B 0,C 180,E1 -24861.166,E2 -24861.166} C_VEL
LIN {X 0,Y 140.517,Z 145.041,A -85,B 0,C 180,E1 -24862.428,E2 -24862.428} C_VEL
LIN {X 0,Y 142.308,Z 148.106,A -85,B 0,C 180,E1 -24863.956,E2 -24863.956} C_VEL
LIN {X 0,Y 144.642,Z 150.456,A -85,B 0,C 180,E1 -24865.651,E2 -24865.651} C_VEL
LIN {X 0,Y 147.105,Z 153.969,A -85,B 0,C 180,E1 -24867.395,E2 -24867.395} C_VEL
LIN {X 0,Y 148.436,Z 155.62,A -85,B 0,C 180,E1 -24868.269,E2 -24868.269} C_VEL
LIN {X 0,Y 151.985,Z 160.67,A -85,B 0,C 180,E1 -24870.499,E2 -24870.499} C_VEL
LIN {X 0,Y 156.561,Z 167.462,A -85,B 0,C 180,E1 -24873.102,E2 -24873.102} C_VEL
LIN {X 0,Y 161.203,Z 175.205,A -85,B 0,C 180,E1 -24875.53,E2 -24875.53} C_VEL
LIN {X 0,Y 167.027,Z 188.634,A -85,B 0,C 180,E1 -24878.481,E2 -24878.481} C_VEL
LIN {X 0,Y 171.379,Z 200.792,A -85,B 0,C 180,E1 -24880.59,E2 -24880.59} C_VEL
LIN {X 0,Y 172.758,Z 205.061,A -85,B 0,C 180,E1 -24881.247,E2 -24881.247} C_VEL
LIN {X 0,Y 168.264,Z 270.272,A -85,B 0,C 180,E1 -24883.66,E2 -24883.66} C_VEL
LIN {X 0,Y 166.399,Z 284.393,A -85,B 0,C 180,E1 -24884.548,E2 -24884.548} C_VEL
LIN {X 0,Y 163.763,Z 297.958,A -85,B 0,C 180,E1 -24885.788,E2 -24885.788} C_VEL
LIN {X 0,Y 160.307,Z 312.132,A -85,B 0,C 180,E1 -24887.625,E2 -24887.625} C_VEL
LIN {X 0,Y 156.417,Z 324.997,A -85,B 0,C 180,E1 -24889.841,E2 -24889.841} C_VEL
LIN {X 0,Y 153.513,Z 333.947,A -85,B 0,C 180,E1 -24891.831,E2 -24891.831} C_VEL
LIN {X 0,Y 150.927,Z 340.769,A -85,B 0,C 180,E1 -24893.584,E2 -24893.584} C_VEL
LIN {X 0,Y 147.095,Z 350.607,A -85,B 0,C 180,E1 -24896.675,E2 -24896.675} C_VEL
LIN {X 0,Y 143.146,Z 360.442,A -85,B 0,C 180,E1 -24900.601,E2 -24900.601} C_VEL
LIN {X 0,Y 139.759,Z 368.828,A -85,B 0,C 180,E1 -24904.862,E2 -24904.862} C_VEL
LIN {X 0,Y 136.924,Z 376.346,A -85,B 0,C 180,E1 -24909.734,E2 -24909.734} C_VEL
LIN {X 0,Y 135.559,Z 380.344,A -85,B 0,C 180,E1 -24912.94,E2 -24912.94} C_VEL
LIN {X 0,Y 134.144,Z 382.82,A -85,B 0,C 180,E1 -24915.143,E2 -24915.143} C_VEL
LIN {X 0,Y 130.43,Z 386.251,A -85,B 0,C 180,E1 -24918.836,E2 -24918.836} C_VEL
LIN {X 0,Y 127.611,Z 388.572,A -85,B 0,C 180,E1 -24921.995,E2 -24921.995} C_VEL
LIN {X 0,Y 126.423,Z 390.132,A -85,B 0,C 180,E1 -24924.533,E2 -24924.533} C_VEL
LIN {X 0,Y 126.317,Z 390.592,A -85,B 0,C 180,E1 -24925.405,E2 -24925.405} C_VEL
LIN {X 0,Y 126.464,Z 392.746,A -85,B 0,C 180,E1 -24930.005,E2 -24930.005} C_VEL
LIN {X 0,Y 126.388,Z 393.763,A -85,B 0,C 180,E1 -24933.192,E2 -24933.192} C_VEL
LIN {X 0,Y 126.732,Z 394.788,A -85,B 0,C 180,E1 -24939.581,E2 -24939.581} C_VEL
LIN {X 0,Y 128.253,Z 394.517,A -85,B 0,C 180,E1 -24945.906,E2 -24945.906} C_VEL
LIN {X 0,Y 131.272,Z 392.962,A -85,B 0,C 180,E1 -24952.014,E2 -24952.014} C_VEL
LIN {X 0,Y 135.628,Z 390.091,A -85,B 0,C 180,E1 -24957.803,E2 -24957.803} C_VEL
LIN {X 0,Y 141.248,Z 385.826,A -85,B 0,C 180,E1 -24963.188,E2 -24963.188} C_VEL
LIN {X 0,Y 148.103,Z 380.044,A -85,B 0,C 180,E1 -24968.094,E2 -24968.094} C_VEL
LIN {X 0,Y 154.982,Z 373.573,A -85,B 0,C 180,E1 -24971.985,E2 -24971.985} C_VEL
LIN {X 0,Y 162.641,Z 365.577,A -85,B 0,C 180,E1 -24975.484,E2 -24975.484} C_VEL
LIN {X 0,Y 169.954,Z 356.732,A -85,B 0,C 180,E1 -24978.424,E2 -24978.424} C_VEL
LIN {X 0,Y 176.887,Z 347.269,A -85,B 0,C 180,E1 -24980.789,E2 -24980.789} C_VEL
LIN {X 0,Y 183.994,Z 336.146,A -85,B 0,C 180,E1 -24982.883,E2 -24982.883} C_VEL
LIN {X 0,Y 190.585,Z 323.749,A -85,B 0,C 180,E1 -24984.679,E2 -24984.679} C_VEL
LIN {X 0,Y 196.112,Z 311.46,A -85,B 0,C 180,E1 -24985.972,E2 -24985.972} C_VEL
LIN {X 0,Y 200.69,Z 298.927,A -85,B 0,C 180,E1 -24986.963,E2 -24986.963} C_VEL
LIN {X 0,Y 204.492,Z 285.335,A -85,B 0,C 180,E1 -24987.764,E2 -24987.764} C_VEL
LIN {X 0,Y 207.186,Z 271.572,A -85,B 0,C 180,E1 -24988.343,E2 -24988.343} C_VEL
LIN {X 0,Y 209.5,Z 250.518,A -85,B 0,C 180,E1 -24988.937,E2 -24988.937} C_VEL
LIN {X 0,Y 210.538,Z 239.507,A -85,B 0,C 180,E1 -24989.228,E2 -24989.228} C_VEL
LIN {X 0,Y 207.178,Z 230.519,A -85,B 0,C 180,E1 -24992.312,E2 -24992.312} C_VEL
LIN {X 0,Y 204.111,Z 223.152,A -85,B 0,C 180,E1 -24995.589,E2 -24995.589} C_VEL
LIN {X 0,Y 202.514,Z 219.737,A -85,B 0,C 180,E1 -24997.552,E2 -24997.552} C_VEL
LIN {X 0,Y 200.623,Z 215.609,A -85,B 0,C 180,E1 -25000.338,E2 -25000.338} C_VEL
LIN {X 0,Y 198.847,Z 212.18,A -85,B 0,C 180,E1 -25003.808,E2 -25003.808} C_VEL
LIN {X 0,Y 197.125,Z 208.038,A -85,B 0,C 180,E1 -25011.795,E2 -25011.795} C_VEL
LIN {X 0,Y 197.258,Z 208.534,A -85,B 0,C 180,E1 -25014.622,E2 -25014.622} C_VEL
LIN {X 0,Y 199.354,Z 212.646,A -85,B 0,C 180,E1 -25021.622,E2 -25021.622} C_VEL
LIN {X 0,Y 201.53,Z 216.801,A -85,B 0,C 180,E1 -25025.39,E2 -25025.39} C_VEL
LIN {X 0,Y 203.824,Z 220.893,A -85,B 0,C 180,E1 -25028.298,E2 -25028.298} C_VEL
LIN {X 0,Y 206.966,Z 226.652,A -85,B 0,C 180,E1 -25031.563,E2 -25031.563} C_VEL
LIN {X 0,Y 210.716,Z 234.224,A -85,B 0,C 180,E1 -25034.85,E2 -25034.85} C_VEL
LIN {X 0,Y 210.976,Z 234.903,A -85,B 0,C 180,E1 -25035.07,E2 -25035.07} C_VEL
LIN {X 0,Y 207.815,Z 265.503,A -85,B 0,C 180,E1 -25035.892,E2 -25035.892} C_VEL
LIN {X 0,Y 205.043,Z 280.179,A -85,B 0,C 180,E1 -25036.526,E2 -25036.526} C_VEL
LIN {X 0,Y 201.52,Z 293.075,A -85,B 0,C 180,E1 -25037.303,E2 -25037.303} C_VEL
LIN {X 0,Y 196.894,Z 306.407,A -85,B 0,C 180,E1 -25038.472,E2 -25038.472} C_VEL
LIN {X 0,Y 191.541,Z 318.75,A -85,B 0,C 180,E1 -25039.902,E2 -25039.902} C_VEL
LIN {X 0,Y 185.277,Z 330.612,A -85,B 0,C 180,E1 -25041.66,E2 -25041.66} C_VEL
LIN {X 0,Y 178.36,Z 341.693,A -85,B 0,C 180,E1 -25043.821,E2 -25043.821} C_VEL
LIN {X 0,Y 171.116,Z 351.633,A -85,B 0,C 180,E1 -25046.384,E2 -25046.384} C_VEL
LIN {X 0,Y 163.464,Z 360.688,A -85,B 0,C 180,E1 -25049.461,E2 -25049.461} C_VEL
LIN {X 0,Y 157.21,Z 367.307,A -85,B 0,C 180,E1 -25052.431,E2 -25052.431} C_VEL
LIN {X 0,Y 151.364,Z 372.826,A -85,B 0,C 180,E1 -25055.649,E2 -25055.649} C_VEL
LIN {X 0,Y 145.616,Z 377.732,A -85,B 0,C 180,E1 -25059.441,E2 -25059.441} C_VEL
LIN {X 0,Y 140.496,Z 381.62,A -85,B 0,C 180,E1 -25063.498,E2 -25063.498} C_VEL
LIN {X 0,Y 136.108,Z 384.582,A -85,B 0,C 180,E1 -25067.83,E2 -25067.83} C_VEL
LIN {X 0,Y 131.508,Z 387.098,A -85,B 0,C 180,E1 -25073.99,E2 -25073.99} C_VEL
LIN {X 0,Y 128.315,Z 388.135,A -85,B 0,C 180,E1 -25080.461,E2 -25080.461} C_VEL
LIN {X 0,Y 126.516,Z 387.732,A -85,B 0,C 180,E1 -25087.112,E2 -25087.112} C_VEL
LIN {X 0,Y 126.047,Z 386.758,A -85,B 0,C 180,E1 -25091.379,E2 -25091.379} C_VEL
LIN {X 0,Y 125.94,Z 384.471,A -85,B 0,C 180,E1 -25097.097,E2 -25097.097} C_VEL
LIN {X 0,Y 126.575,Z 381.589,A -85,B 0,C 180,E1 -25102.016,E2 -25102.016} C_VEL
LIN {X 0,Y 127.668,Z 377.888,A -85,B 0,C 180,E1 -25106.84,E2 -25106.84} C_VEL
LIN {X 0,Y 129.218,Z 373.255,A -85,B 0,C 180,E1 -25111.554,E2 -25111.554} C_VEL
LIN {X 0,Y 131.925,Z 366.549,A -85,B 0,C 180,E1 -25116.88,E2 -25116.88} C_VEL
LIN {X 0,Y 135.561,Z 358.193,A -85,B 0,C 180,E1 -25121.964,E2 -25121.964} C_VEL
LIN {X 0,Y 139.63,Z 348.766,A -85,B 0,C 180,E1 -25126.393,E2 -25126.393} C_VEL
LIN {X 0,Y 143.491,Z 338.962,A -85,B 0,C 180,E1 -25130.046,E2 -25130.046} C_VEL
LIN {X 0,Y 147.709,Z 328.29,A -85,B 0,C 180,E1 -25133.108,E2 -25133.108} C_VEL
LIN {X 0,Y 151.741,Z 316.669,A -85,B 0,C 180,E1 -25135.731,E2 -25135.731} C_VEL
LIN {X 0,Y 155.525,Z 303.916,A -85,B 0,C 180,E1 -25137.954,E2 -25137.954} C_VEL
LIN {X 0,Y 158.688,Z 290.746,A -85,B 0,C 180,E1 -25139.697,E2 -25139.697} C_VEL
LIN {X 0,Y 161.272,Z 276.544,A -85,B 0,C 180,E1 -25141.069,E2 -25141.069} C_VEL
LIN {X 0,Y 163.085,Z 262.288,A -85,B 0,C 180,E1 -25141.965,E2 -25141.965} C_VEL
LIN {X 0,Y 167.673,Z 200.682,A -85,B 0,C 180,E1 -25144.204,E2 -25144.204} C_VEL
LIN {X 0,Y 162.197,Z 188.935,A -85,B 0,C 180,E1 -25146.822,E2 -25146.822} C_VEL
LIN {X 0,Y 155.907,Z 177.38,A -85,B 0,C 180,E1 -25150.102,E2 -25150.102} C_VEL
LIN {X 0,Y 149.998,Z 167.9,A -85,B 0,C 180,E1 -25153.554,E2 -25153.554} C_VEL
LIN {X 0,Y 146.943,Z 163.574,A -85,B 0,C 180,E1 -25155.503,E2 -25155.503} C_VEL
LIN {X 0,Y 144.387,Z 159.941,A -85,B 0,C 180,E1 -25157.274,E2 -25157.274} C_VEL
LIN {X 0,Y 141.338,Z 155.81,A -85,B 0,C 180,E1 -25159.572,E2 -25159.572} C_VEL
LIN {X 0,Y 138.704,Z 152.529,A -85,B 0,C 180,E1 -25161.738,E2 -25161.738} C_VEL
LIN {X 0,Y 137.851,Z 151.151,A -85,B 0,C 180,E1 -25162.525,E2 -25162.525} C_VEL
LIN {X 0,Y 135.316,Z 148.867,A -85,B 0,C 180,E1 -25164.831,E2 -25164.831} C_VEL
LIN {X 0,Y 133.57,Z 145.812,A -85,B 0,C 180,E1 -25166.775,E2 -25166.775} C_VEL
LIN {X 0,Y 130.803,Z 143.92,A -85,B 0,C 180,E1 -25169.878,E2 -25169.878} C_VEL
LIN {X 0,Y 129.494,Z 141.665,A -85,B 0,C 180,E1 -25171.771,E2 -25171.771} C_VEL
LIN {X 0,Y 129.062,Z 139.985,A -85,B 0,C 180,E1 -25172.66,E2 -25172.66} C_VEL
LIN {X 0,Y 129.113,Z 140.024,A -85,B 0,C 180,E1 -25177.71,E2 -25177.71} C_VEL
LIN {X 0,Y 129.169,Z 140.011,A -85,B 0,C 180,E1 -25180.958,E2 -25180.958} C_VEL
LIN {X 0,Y 129.404,Z 139.989,A -85,B 0,C 180,E1 -25187.824,E2 -25187.824} C_VEL
LIN {X 0,Y 129.516,Z 139.946,A -85,B 0,C 180,E1 -25190.642,E2 -25190.642} C_VEL
LIN {X 0,Y 130.08,Z 139.902,A -85,B 0,C 180,E1 -25200.01,E2 -25200.01} C_VEL
LIN {X 0,Y 129.511,Z 139.976,A -85,B 0,C 180,E1 -25209.379,E2 -25209.379} C_VEL
LIN {X 0,Y 129.476,Z 140.094,A -85,B 0,C 180,E1 -25211.565,E2 -25211.565} C_VEL
LIN {X 0,Y 130.215,Z 142.615,A -85,B 0,C 180,E1 -25212.874,E2 -25212.874} C_VEL
LIN {X 0,Y 132.071,Z 144.867,A -85,B 0,C 180,E1 -25215.243,E2 -25215.243} C_VEL
LIN {X 0,Y 133.989,Z 145.971,A -85,B 0,C 180,E1 -25217.268,E2 -25217.268} C_VEL
LIN {X 0,Y 135.552,Z 148.916,A -85,B 0,C 180,E1 -25219.016,E2 -25219.016} C_VEL
LIN {X 0,Y 138.165,Z 151.529,A -85,B 0,C 180,E1 -25221.394,E2 -25221.394} C_VEL
LIN {X 0,Y 140.588,Z 155.097,A -85,B 0,C 180,E1 -25223.493,E2 -25223.493} C_VEL
LIN {X 0,Y 142.071,Z 156.731,A -85,B 0,C 180,E1 -25224.63,E2 -25224.63} C_VEL
LIN {X 0,Y 144.93,Z 160.536,A -85,B 0,C 180,E1 -25226.725,E2 -25226.725} C_VEL
LIN {X 0,Y 150.719,Z 169.045,A -85,B 0,C 180,E1 -25230.528,E2 -25230.528} C_VEL
LIN {X 0,Y 156.988,Z 179.357,A -85,B 0,C 180,E1 -25234.117,E2 -25234.117} C_VEL
LIN {X 0,Y 162.577,Z 192.693,A -85,B 0,C 180,E1 -25237.177,E2 -25237.177} C_VEL
LIN {X 0,Y 166.482,Z 203.972,A -85,B 0,C 180,E1 -25239.222,E2 -25239.222} C_VEL
LIN {X 0,Y 167.403,Z 206.966,A -85,B 0,C 180,E1 -25239.701,E2 -25239.701} C_VEL
LIN {X 0,Y 162.83,Z 270.234,A -85,B 0,C 180,E1 -25242.078,E2 -25242.078} C_VEL
LIN {X 0,Y 160.9,Z 284.332,A -85,B 0,C 180,E1 -25242.983,E2 -25242.983} C_VEL
LIN {X 0,Y 158.168,Z 297.862,A -85,B 0,C 180,E1 -25244.24,E2 -25244.24} C_VEL
LIN {X 0,Y 154.578,Z 312.017,A -85,B 0,C 180,E1 -25246.11,E2 -25246.11} C_VEL
LIN {X 0,Y 150.463,Z 325.021,A -85,B 0,C 180,E1 -25248.397,E2 -25248.397} C_VEL
LIN {X 0,Y 147.487,Z 333.806,A -85,B 0,C 180,E1 -25250.411,E2 -25250.411} C_VEL
LIN {X 0,Y 144.788,Z 340.623,A -85,B 0,C 180,E1 -25252.212,E2 -25252.212} C_VEL
LIN {X 0,Y 140.38,Z 351.356,A -85,B 0,C 180,E1 -25255.726,E2 -25255.726} C_VEL
LIN {X 0,Y 136.288,Z 361.037,A -85,B 0,C 180,E1 -25259.821,E2 -25259.821} C_VEL
LIN {X 0,Y 132.982,Z 368.757,A -85,B 0,C 180,E1 -25263.972,E2 -25263.972} C_VEL
LIN {X 0,Y 129.859,Z 376.681,A -85,B 0,C 180,E1 -25269.409,E2 -25269.409} C_VEL
LIN {X 0,Y 127.963,Z 381.949,A -85,B 0,C 180,E1 -25274.066,E2 -25274.066} C_VEL
LIN {X 0,Y 126.913,Z 386.231,A -85,B 0,C 180,E1 -25278.829,E2 -25278.829} C_VEL
LIN {X 0,Y 126.416,Z 389.617,A -85,B 0,C 180,E1 -25283.621,E2 -25283.621} C_VEL
LIN {X 0,Y 126.317,Z 390.592,A -85,B 0,C 180,E1 -25285.405,E2 -25285.405} C_VEL
LIN {X 0,Y 125.582,Z 391.879,A -85,B 0,C 180,E1 -25288.002,E2 -25288.002} C_VEL
LIN {X 0,Y 123.946,Z 392.849,A -85,B 0,C 180,E1 -25290.591,E2 -25290.591} C_VEL
LIN {X 0,Y 120.349,Z 394.101,A -85,B 0,C 180,E1 -25295.961,E2 -25295.961} C_VEL
LIN {X 0,Y 119.587,Z 394.449,A -85,B 0,C 180,E1 -25298.805,E2 -25298.805} C_VEL
LIN {X 0,Y 119.644,Z 394.527,A -85,B 0,C 180,E1 -25299.763,E2 -25299.763} C_VEL
LIN {X 0,Y 120.417,Z 394.636,A -85,B 0,C 180,E1 -25303.505,E2 -25303.505} C_VEL
LIN {X 0,Y 122.826,Z 393.799,A -85,B 0,C 180,E1 -25310.084,E2 -25310.084} C_VEL
LIN {X 0,Y 126.842,Z 391.671,A -85,B 0,C 180,E1 -25316.317,E2 -25316.317} C_VEL
LIN {X 0,Y 132.168,Z 388.198,A -85,B 0,C 180,E1 -25322.128,E2 -25322.128} C_VEL
LIN {X 0,Y 138.807,Z 383.278,A -85,B 0,C 180,E1 -25327.419,E2 -25327.419} C_VEL
LIN {X 0,Y 146.58,Z 376.769,A -85,B 0,C 180,E1 -25332.168,E2 -25332.168} C_VEL
LIN {X 0,Y 154.264,Z 369.562,A -85,B 0,C 180,E1 -25335.857,E2 -25335.857} C_VEL
LIN {X 0,Y 162.551,Z 360.693,A -85,B 0,C 180,E1 -25339.173,E2 -25339.173} C_VEL
LIN {X 0,Y 169.915,Z 351.456,A -85,B 0,C 180,E1 -25341.807,E2 -25341.807} C_VEL
LIN {X 0,Y 177.784,Z 340.212,A -85,B 0,C 180,E1 -25344.139,E2 -25344.139} C_VEL
LIN {X 0,Y 184.556,Z 328.815,A -85,B 0,C 180,E1 -25345.924,E2 -25345.924} C_VEL
LIN {X 0,Y 190.136,Z 317.772,A -85,B 0,C 180,E1 -25347.241,E2 -25347.241} C_VEL
LIN {X 0,Y 195.102,Z 305.939,A -85,B 0,C 180,E1 -25348.328,E2 -25348.328} C_VEL
LIN {X 0,Y 199.582,Z 292.574,A -85,B 0,C 180,E1 -25349.222,E2 -25349.222} C_VEL
LIN {X 0,Y 203.153,Z 278.3,A -85,B 0,C 180,E1 -25349.872,E2 -25349.872} C_VEL
LIN {X 0,Y 205.385,Z 263.824,A -85,B 0,C 180,E1 -25350.382,E2 -25350.382} C_VEL
LIN {X 0,Y 207.438,Z 242.871,A -85,B 0,C 180,E1 -25350.949,E2 -25350.949} C_VEL
LIN {X 0,Y 204.625,Z 235.06,A -85,B 0,C 180,E1 -25353.812,E2 -25353.812} C_VEL
LIN {X 0,Y 202.059,Z 228.535,A -85,B 0,C 180,E1 -25356.855,E2 -25356.855} C_VEL
LIN {X 0,Y 199.519,Z 222.676,A -85,B 0,C 180,E1 -25360.605,E2 -25360.605} C_VEL
LIN {X 0,Y 197.874,Z 219.196,A -85,B 0,C 180,E1 -25363.966,E2 -25363.966} C_VEL
LIN {X 0,Y 196.226,Z 215.218,A -85,B 0,C 180,E1 -25371.757,E2 -25371.757} C_VEL
LIN {X 0,Y 196.375,Z 215.641,A -85,B 0,C 180,E1 -25374.682,E2 -25374.682} C_VEL
LIN {X 0,Y 198.248,Z 219.591,A -85,B 0,C 180,E1 -25381.237,E2 -25381.237} C_VEL
LIN {X 0,Y 200.253,Z 223.628,A -85,B 0,C 180,E1 -25384.927,E2 -25384.927} C_VEL
LIN {X 0,Y 202.363,Z 227.573,A -85,B 0,C 180,E1 -25387.741,E2 -25387.741} C_VEL
LIN {X 0,Y 205.337,Z 233.401,A -85,B 0,C 180,E1 -25391,E2 -25391} C_VEL
LIN {X 0,Y 207.863,Z 238.668,A -85,B 0,C 180,E1 -25393.372,E2 -25393.372} C_VEL
LIN {X 0,Y 204.967,Z 265.718,A -85,B 0,C 180,E1 -25394.094,E2 -25394.094} C_VEL
LIN {X 0,Y 202.1,Z 280.465,A -85,B 0,C 180,E1 -25394.711,E2 -25394.711} C_VEL
LIN {X 0,Y 198.301,Z 293.927,A -85,B 0,C 180,E1 -25395.507,E2 -25395.507} C_VEL
LIN {X 0,Y 193.698,Z 306.737,A -85,B 0,C 180,E1 -25396.614,E2 -25396.614} C_VEL
LIN {X 0,Y 188.388,Z 318.594,A -85,B 0,C 180,E1 -25397.946,E2 -25397.946} C_VEL
LIN {X 0,Y 181.938,Z 330.503,A -85,B 0,C 180,E1 -25399.675,E2 -25399.675} C_VEL
LIN {X 0,Y 175.235,Z 340.955,A -85,B 0,C 180,E1 -25401.654,E2 -25401.654} C_VEL
LIN {X 0,Y 167.652,Z 351.091,A -85,B 0,C 180,E1 -25404.155,E2 -25404.155} C_VEL
LIN {X 0,Y 159.877,Z 360.047,A -85,B 0,C 180,E1 -25407.099,E2 -25407.099} C_VEL
LIN {X 0,Y 152.365,Z 367.646,A -85,B 0,C 180,E1 -25410.479,E2 -25410.479} C_VEL
LIN {X 0,Y 144.948,Z 374.223,A -85,B 0,C 180,E1 -25414.479,E2 -25414.479} C_VEL
LIN {X 0,Y 138.988,Z 378.922,A -85,B 0,C 180,E1 -25418.387,E2 -25418.387} C_VEL
LIN {X 0,Y 132.682,Z 383.218,A -85,B 0,C 180,E1 -25423.503,E2 -25423.503} C_VEL
LIN {X 0,Y 127.833,Z 386.029,A -85,B 0,C 180,E1 -25428.715,E2 -25428.715} C_VEL
LIN {X 0,Y 123.416,Z 387.923,A -85,B 0,C 180,E1 -25435.282,E2 -25435.282} C_VEL
LIN {X 0,Y 120.546,Z 388.346,A -85,B 0,C 180,E1 -25442.193,E2 -25442.193} C_VEL
LIN {X 0,Y 119.101,Z 387.337,A -85,B 0,C 180,E1 -25449.26,E2 -25449.26} C_VEL
LIN {X 0,Y 118.848,Z 386.301,A -85,B 0,C 180,E1 -25452.797,E2 -25452.797} C_VEL
LIN {X 0,Y 119.084,Z 383.165,A -85,B 0,C 180,E1 -25459.797,E2 -25459.797} C_VEL
LIN {X 0,Y 119.974,Z 380.054,A -85,B 0,C 180,E1 -25464.637,E2 -25464.637} C_VEL
LIN {X 0,Y 121.449,Z 375.616,A -85,B 0,C 180,E1 -25469.995,E2 -25469.995} C_VEL
LIN {X 0,Y 123.48,Z 370.417,A -85,B 0,C 180,E1 -25474.893,E2 -25474.893} C_VEL
LIN {X 0,Y 126.86,Z 362.967,A -85,B 0,C 180,E1 -25480.368,E2 -25480.368} C_VEL
LIN {X 0,Y 130.487,Z 355.164,A -85,B 0,C 180,E1 -25484.818,E2 -25484.818} C_VEL
LIN {X 0,Y 134.694,Z 345.798,A -85,B 0,C 180,E1 -25489.028,E2 -25489.028} C_VEL
LIN {X 0,Y 138.869,Z 335.476,A -85,B 0,C 180,E1 -25492.695,E2 -25492.695} C_VEL
LIN {X 0,Y 143.447,Z 323.991,A -85,B 0,C 180,E1 -25495.769,E2 -25495.769} C_VEL
LIN {X 0,Y 147.802,Z 311.295,A -85,B 0,C 180,E1 -25498.387,E2 -25498.387} C_VEL
LIN {X 0,Y 151.33,Z 298.994,A -85,B 0,C 180,E1 -25500.33,E2 -25500.33} C_VEL
LIN {X 0,Y 154.336,Z 285.484,A -85,B 0,C 180,E1 -25501.958,E2 -25501.958} C_VEL
LIN {X 0,Y 156.713,Z 271.359,A -85,B 0,C 180,E1 -25503.145,E2 -25503.145} C_VEL
LIN {X 0,Y 158.305,Z 257.307,A -85,B 0,C 180,E1 -25503.874,E2 -25503.874} C_VEL
LIN {X 0,Y 162.426,Z 202.927,A -85,B 0,C 180,E1 -25505.851,E2 -25505.851} C_VEL
LIN {X 0,Y 156.484,Z 190.301,A -85,B 0,C 180,E1 -25508.954,E2 -25508.954} C_VEL
LIN {X 0,Y 150.914,Z 180.144,A -85,B 0,C 180,E1 -25512.159,E2 -25512.159} C_VEL
LIN {X 0,Y 145.003,Z 170.581,A -85,B 0,C 180,E1 -25515.982,E2 -25515.982} C_VEL
LIN {X 0,Y 141.191,Z 165.307,A -85,B 0,C 180,E1 -25518.752,E2 -25518.752} C_VEL
LIN {X 0,Y 138.768,Z 161.886,A -85,B 0,C 180,E1 -25520.717,E2 -25520.717} C_VEL
LIN {X 0,Y 136.057,Z 158.198,A -85,B 0,C 180,E1 -25523.138,E2 -25523.138} C_VEL
LIN {X 0,Y 134.834,Z 156.904,A -85,B 0,C 180,E1 -25524.285,E2 -25524.285} C_VEL
LIN {X 0,Y 132.468,Z 153.987,A -85,B 0,C 180,E1 -25526.753,E2 -25526.753} C_VEL
LIN {X 0,Y 131.655,Z 152.472,A -85,B 0,C 180,E1 -25527.749,E2 -25527.749} C_VEL
LIN {X 0,Y 128.915,Z 150.238,A -85,B 0,C 180,E1 -25531.083,E2 -25531.083} C_VEL
LIN {X 0,Y 127.511,Z 147.541,A -85,B 0,C 180,E1 -25533.342,E2 -25533.342} C_VEL
LIN {X 0,Y 127.272,Z 146.882,A -85,B 0,C 180,E1 -25533.796,E2 -25533.796} C_VEL
LIN {X 0,Y 124.256,Z 145.195,A -85,B 0,C 180,E1 -25539.325,E2 -25539.325} C_VEL
LIN {X 0,Y 122.432,Z 141.949,A -85,B 0,C 180,E1 -25545.891,E2 -25545.891} C_VEL
LIN {X 0,Y 122.351,Z 140.866,A -85,B 0,C 180,E1 -25547.532,E2 -25547.532} C_VEL
LIN {X 0,Y 122.442,Z 140.833,A -85,B 0,C 180,E1 -25550.096,E2 -25550.096} C_VEL
LIN {X 0,Y 122.916,Z 140.904,A -85,B 0,C 180,E1 -25559.192,E2 -25559.192} C_VEL
LIN {X 0,Y 123.129,Z 141.553,A -85,B 0,C 180,E1 -25560.215,E2 -25560.215} C_VEL
LIN {X 0,Y 123.656,Z 143.605,A -85,B 0,C 180,E1 -25562.454,E2 -25562.454} C_VEL
LIN {X 0,Y 125.714,Z 145.981,A -85,B 0,C 180,E1 -25567.236,E2 -25567.236} C_VEL
LIN {X 0,Y 127.693,Z 147.073,A -85,B 0,C 180,E1 -25570.441,E2 -25570.441} C_VEL
LIN {X 0,Y 128.995,Z 149.988,A -85,B 0,C 180,E1 -25572.598,E2 -25572.598} C_VEL
LIN {X 0,Y 131.349,Z 152.191,A -85,B 0,C 180,E1 -25575.527,E2 -25575.527} C_VEL
LIN {X 0,Y 132.135,Z 152.984,A -85,B 0,C 180,E1 -25576.423,E2 -25576.423} C_VEL
LIN {X 0,Y 134.434,Z 156.395,A -85,B 0,C 180,E1 -25578.957,E2 -25578.957} C_VEL
LIN {X 0,Y 135.915,Z 157.969,A -85,B 0,C 180,E1 -25580.364,E2 -25580.364} C_VEL
LIN {X 0,Y 138.558,Z 161.684,A -85,B 0,C 180,E1 -25582.751,E2 -25582.751} C_VEL
LIN {X 0,Y 139.746,Z 163.261,A -85,B 0,C 180,E1 -25583.733,E2 -25583.733} C_VEL
LIN {X 0,Y 143.137,Z 168.053,A -85,B 0,C 180,E1 -25586.341,E2 -25586.341} C_VEL
LIN {X 0,Y 147.258,Z 174.18,A -85,B 0,C 180,E1 -25589.174,E2 -25589.174} C_VEL
LIN {X 0,Y 153.166,Z 184.231,A -85,B 0,C 180,E1 -25592.818,E2 -25592.818} C_VEL
LIN {X 0,Y 158.606,Z 197.796,A -85,B 0,C 180,E1 -25596.021,E2 -25596.021} C_VEL
LIN {X 0,Y 162.177,Z 208.827,A -85,B 0,C 180,E1 -25598.052,E2 -25598.052} C_VEL
LIN {X 0,Y 157.517,Z 270.417,A -85,B 0,C 180,E1 -25600.405,E2 -25600.405} C_VEL
LIN {X 0,Y 155.53,Z 284.271,A -85,B 0,C 180,E1 -25601.308,E2 -25601.308} C_VEL
LIN {X 0,Y 152.694,Z 297.766,A -85,B 0,C 180,E1 -25602.578,E2 -25602.578} C_VEL
LIN {X 0,Y 148.965,Z 311.902,A -85,B 0,C 180,E1 -25604.479,E2 -25604.479} C_VEL
LIN {X 0,Y 144.915,Z 324.252,A -85,B 0,C 180,E1 -25606.685,E2 -25606.685} C_VEL
LIN {X 0,Y 141.558,Z 333.664,A -85,B 0,C 180,E1 -25608.871,E2 -25608.871} C_VEL
LIN {X 0,Y 138.728,Z 340.474,A -85,B 0,C 180,E1 -25610.715,E2 -25610.715} C_VEL
LIN {X 0,Y 134.527,Z 350.299,A -85,B 0,C 180,E1 -25614.01,E2 -25614.01} C_VEL
LIN {X 0,Y 130.107,Z 360.115,A -85,B 0,C 180,E1 -25618.225,E2 -25618.225} C_VEL
LIN {X 0,Y 126.249,Z 368.671,A -85,B 0,C 180,E1 -25622.978,E2 -25622.978} C_VEL
LIN {X 0,Y 123.153,Z 376,A -85,B 0,C 180,E1 -25628.232,E2 -25628.232} C_VEL
LIN {X 0,Y 121.095,Z 381.362,A -85,B 0,C 180,E1 -25633.136,E2 -25633.136} C_VEL
LIN {X 0,Y 119.652,Z 386.992,A -85,B 0,C 180,E1 -25639.856,E2 -25639.856} C_VEL
LIN {X 0,Y 119.225,Z 390.346,A -85,B 0,C 180,E1 -25645.417,E2 -25645.417} C_VEL
LIN {X 0,Y 119.379,Z 392.416,A -85,B 0,C 180,E1 -25650.005,E2 -25650.005} C_VEL
LIN {X 0,Y 119.295,Z 393.471,A -85,B 0,C 180,E1 -25653.382,E2 -25653.382} C_VEL
LIN {X 0,Y 119.644,Z 394.527,A -85,B 0,C 180,E1 -25659.763,E2 -25659.763} C_VEL
LIN {X 0,Y 119.525,Z 394.721,A -85,B 0,C 180,E1 -25662.589,E2 -25662.589} C_VEL
LIN {X 0,Y 118.059,Z 394.492,A -85,B 0,C 180,E1 -25667.319,E2 -25667.319} C_VEL
LIN {X 0,Y 117.29,Z 393.822,A -85,B 0,C 180,E1 -25671.166,E2 -25671.166} C_VEL
LIN {X 0,Y 117.842,Z 393.037,A -85,B 0,C 180,E1 -25674.016,E2 -25674.016} C_VEL
LIN {X 0,Y 118.352,Z 392.722,A -85,B 0,C 180,E1 -25674.929,E2 -25674.929} C_VEL
LIN {X 0,Y 123.171,Z 390.125,A -85,B 0,C 180,E1 -25680.904,E2 -25680.904} C_VEL
LIN {X 0,Y 129.541,Z 386.027,A -85,B 0,C 180,E1 -25686.645,E2 -25686.645} C_VEL
LIN {X 0,Y 137.209,Z 380.421,A -85,B 0,C 180,E1 -25691.755,E2 -25691.755} C_VEL
LIN {X 0,Y 144.724,Z 374.15,A -85,B 0,C 180,E1 -25695.754,E2 -25695.754} C_VEL
LIN {X 0,Y 153.052,Z 366.381,A -85,B 0,C 180,E1 -25699.264,E2 -25699.264} C_VEL
LIN {X 0,Y 160.47,Z 358.322,A -85,B 0,C 180,E1 -25702.035,E2 -25702.035} C_VEL
LIN {X 0,Y 168.335,Z 348.641,A -85,B 0,C 180,E1 -25704.506,E2 -25704.506} C_VEL
LIN {X 0,Y 175.854,Z 337.922,A -85,B 0,C 180,E1 -25706.545,E2 -25706.545} C_VEL
LIN {X 0,Y 182.823,Z 326.105,A -85,B 0,C 180,E1 -25708.274,E2 -25708.274} C_VEL
LIN {X 0,Y 188.623,Z 314.484,A -85,B 0,C 180,E1 -25709.505,E2 -25709.505} C_VEL
LIN {X 0,Y 193.751,Z 301.853,A -85,B 0,C 180,E1 -25710.529,E2 -25710.529} C_VEL
LIN {X 0,Y 198.072,Z 288.231,A -85,B 0,C 180,E1 -25711.331,E2 -25711.331} C_VEL
LIN {X 0,Y 201.178,Z 274.643,A -85,B 0,C 180,E1 -25711.895,E2 -25711.895} C_VEL
LIN {X 0,Y 203.331,Z 258.861,A -85,B 0,C 180,E1 -25712.348,E2 -25712.348} C_VEL
LIN {X 0,Y 204.509,Z 246.411,A -85,B 0,C 180,E1 -25712.717,E2 -25712.717} C_VEL
LIN {X 0,Y 202.177,Z 239.503,A -85,B 0,C 180,E1 -25715.395,E2 -25715.395} C_VEL
LIN {X 0,Y 200.027,Z 233.697,A -85,B 0,C 180,E1 -25718.267,E2 -25718.267} C_VEL
LIN {X 0,Y 198.03,Z 228.917,A -85,B 0,C 180,E1 -25721.597,E2 -25721.597} C_VEL
LIN {X 0,Y 196.692,Z 226.011,A -85,B 0,C 180,E1 -25724.611,E2 -25724.611} C_VEL
LIN {X 0,Y 195.328,Z 222.382,A -85,B 0,C 180,E1 -25731.719,E2 -25731.719} C_VEL
LIN {X 0,Y 195.439,Z 222.555,A -85,B 0,C 180,E1 -25734.229,E2 -25734.229} C_VEL
LIN {X 0,Y 197.11,Z 226.376,A -85,B 0,C 180,E1 -25740.733,E2 -25740.733} C_VEL
LIN {X 0,Y 198.84,Z 230.085,A -85,B 0,C 180,E1 -25744.177,E2 -25744.177} C_VEL
LIN {X 0,Y 201.027,Z 234.497,A -85,B 0,C 180,E1 -25747.315,E2 -25747.315} C_VEL
LIN {X 0,Y 204.078,Z 240.839,A -85,B 0,C 180,E1 -25750.786,E2 -25750.786} C_VEL
LIN {X 0,Y 204.913,Z 242.708,A -85,B 0,C 180,E1 -25751.633,E2 -25751.633} C_VEL
LIN {X 0,Y 202.302,Z 266.038,A -85,B 0,C 180,E1 -25752.246,E2 -25752.246} C_VEL
LIN {X 0,Y 199.418,Z 280.49,A -85,B 0,C 180,E1 -25752.824,E2 -25752.824} C_VEL
LIN {X 0,Y 195.628,Z 293.734,A -85,B 0,C 180,E1 -25753.585,E2 -25753.585} C_VEL
LIN {X 0,Y 190.731,Z 307.026,A -85,B 0,C 180,E1 -25754.693,E2 -25754.693} C_VEL
LIN {X 0,Y 184.707,Z 319.999,A -85,B 0,C 180,E1 -25756.128,E2 -25756.128} C_VEL
LIN {X 0,Y 178.092,Z 331.641,A -85,B 0,C 180,E1 -25757.807,E2 -25757.807} C_VEL
LIN {X 0,Y 171.614,Z 341.308,A -85,B 0,C 180,E1 -25759.617,E2 -25759.617} C_VEL
LIN {X 0,Y 164.637,Z 350.35,A -85,B 0,C 180,E1 -25761.797,E2 -25761.797} C_VEL
LIN {X 0,Y 156.609,Z 359.402,A -85,B 0,C 180,E1 -25764.66,E2 -25764.66} C_VEL
LIN {X 0,Y 148.695,Z 367.129,A -85,B 0,C 180,E1 -25767.954,E2 -25767.954} C_VEL
LIN {X 0,Y 140.788,Z 373.87,A -85,B 0,C 180,E1 -25771.931,E2 -25771.931} C_VEL
LIN {X 0,Y 134.413,Z 378.645,A -85,B 0,C 180,E1 -25775.854,E2 -25775.854} C_VEL
LIN {X 0,Y 128.651,Z 382.401,A -85,B 0,C 180,E1 -25780.105,E2 -25780.105} C_VEL
LIN {X 0,Y 122.211,Z 385.988,A -85,B 0,C 180,E1 -25786.357,E2 -25786.357} C_VEL
LIN {X 0,Y 117.287,Z 388.036,A -85,B 0,C 180,E1 -25793.181,E2 -25793.181} C_VEL
LIN {X 0,Y 113.956,Z 388.579,A -85,B 0,C 180,E1 -25800.431,E2 -25800.431} C_VEL
LIN {X 0,Y 112.163,Z 387.677,A -85,B 0,C 180,E1 -25807.911,E2 -25807.911} C_VEL
LIN {X 0,Y 111.815,Z 386.692,A -85,B 0,C 180,E1 -25811.678,E2 -25811.678} C_VEL
LIN {X 0,Y 111.884,Z 383.663,A -85,B 0,C 180,E1 -25819.133,E2 -25819.133} C_VEL
LIN {X 0,Y 112.886,Z 380.305,A -85,B 0,C 180,E1 -25824.798,E2 -25824.798} C_VEL
LIN {X 0,Y 114.252,Z 376.313,A -85,B 0,C 180,E1 -25829.995,E2 -25829.995} C_VEL
LIN {X 0,Y 116.338,Z 371.203,A -85,B 0,C 180,E1 -25835.194,E2 -25835.194} C_VEL
LIN {X 0,Y 119.839,Z 363.892,A -85,B 0,C 180,E1 -25840.983,E2 -25840.983} C_VEL
LIN {X 0,Y 123.613,Z 356.235,A -85,B 0,C 180,E1 -25845.663,E2 -25845.663} C_VEL
LIN {X 0,Y 128.012,Z 347.051,A -85,B 0,C 180,E1 -25850.063,E2 -25850.063} C_VEL
LIN {X 0,Y 131.886,Z 337.956,A -85,B 0,C 180,E1 -25853.552,E2 -25853.552} C_VEL
LIN {X 0,Y 136.648,Z 326.983,A -85,B 0,C 180,E1 -25856.74,E2 -25856.74} C_VEL
LIN {X 0,Y 141.047,Z 315.021,A -85,B 0,C 180,E1 -25859.47,E2 -25859.47} C_VEL
LIN {X 0,Y 145.227,Z 301.749,A -85,B 0,C 180,E1 -25861.749,E2 -25861.749} C_VEL
LIN {X 0,Y 148.389,Z 289,A -85,B 0,C 180,E1 -25863.402,E2 -25863.402} C_VEL
LIN {X 0,Y 151.076,Z 274.572,A -85,B 0,C 180,E1 -25864.738,E2 -25864.738} C_VEL
LIN {X 0,Y 152.876,Z 261.097,A -85,B 0,C 180,E1 -25865.523,E2 -25865.523} C_VEL
LIN {X 0,Y 157.356,Z 205.951,A -85,B 0,C 180,E1 -25867.542,E2 -25867.542} C_VEL
LIN {X 0,Y 156.465,Z 203.385,A -85,B 0,C 180,E1 -25868.066,E2 -25868.066} C_VEL
LIN {X 0,Y 151.349,Z 192.612,A -85,B 0,C 180,E1 -25871.015,E2 -25871.015} C_VEL
LIN {X 0,Y 146.638,Z 183.951,A -85,B 0,C 180,E1 -25873.979,E2 -25873.979} C_VEL
LIN {X 0,Y 141.768,Z 175.926,A -85,B 0,C 180,E1 -25877.399,E2 -25877.399} C_VEL
LIN {X 0,Y 136.51,Z 168.194,A -85,B 0,C 180,E1 -25881.689,E2 -25881.689} C_VEL
LIN {X 0,Y 133.122,Z 163.66,A -85,B 0,C 180,E1 -25884.938,E2 -25884.938} C_VEL
LIN {X 0,Y 130.483,Z 160.366,A -85,B 0,C 180,E1 -25887.843,E2 -25887.843} C_VEL
LIN {X 0,Y 129.676,Z 159.028,A -85,B 0,C 180,E1 -25888.876,E2 -25888.876} C_VEL
LIN {X 0,Y 127.044,Z 156.478,A -85,B 0,C 180,E1 -25892.383,E2 -25892.383} C_VEL
LIN {X 0,Y 125.701,Z 153.746,A -85,B 0,C 180,E1 -25894.779,E2 -25894.779} C_VEL
LIN {X 0,Y 122.704,Z 151.615,A -85,B 0,C 180,E1 -25901.001,E2 -25901.001} C_VEL
LIN {X 0,Y 121.345,Z 148.293,A -85,B 0,C 180,E1 -25907.427,E2 -25907.427} C_VEL
LIN {X 0,Y 121.255,Z 147.867,A -85,B 0,C 180,E1 -25908.461,E2 -25908.461} C_VEL
LIN {X 0,Y 121.914,Z 147.952,A -85,B 0,C 180,E1 -25918.772,E2 -25918.772} C_VEL
LIN {X 0,Y 122.667,Z 150.778,A -85,B 0,C 180,E1 -25922.268,E2 -25922.268} C_VEL
LIN {X 0,Y 124.819,Z 153.09,A -85,B 0,C 180,E1 -25927.289,E2 -25927.289} C_VEL
LIN {X 0,Y 126.082,Z 153.898,A -85,B 0,C 180,E1 -25929.434,E2 -25929.434} C_VEL
LIN {X 0,Y 127.671,Z 157.011,A -85,B 0,C 180,E1 -25932.125,E2 -25932.125} C_VEL
LIN {X 0,Y 130.214,Z 159.516,A -85,B 0,C 180,E1 -25935.386,E2 -25935.386} C_VEL
LIN {X 0,Y 132.584,Z 162.979,A -85,B 0,C 180,E1 -25938.14,E2 -25938.14} C_VEL
LIN {X 0,Y 133.71,Z 164.316,A -85,B 0,C 180,E1 -25939.288,E2 -25939.288} C_VEL
LIN {X 0,Y 137.327,Z 169.486,A -85,B 0,C 180,E1 -25942.682,E2 -25942.682} C_VEL
LIN {X 0,Y 140.86,Z 174.693,A -85,B 0,C 180,E1 -25945.56,E2 -25945.56} C_VEL
LIN {X 0,Y 144.745,Z 180.817,A -85,B 0,C 180,E1 -25948.376,E2 -25948.376} C_VEL
LIN {X 0,Y 149.428,Z 189.125,A -85,B 0,C 180,E1 -25951.455,E2 -25951.455} C_VEL
LIN {X 0,Y 154.239,Z 201.641,A -85,B 0,C 180,E1 -25954.526,E2 -25954.526} C_VEL
LIN {X 0,Y 157.066,Z 210.567,A -85,B 0,C 180,E1 -25956.277,E2 -25956.277} C_VEL
LIN {X 0,Y 152.488,Z 269.493,A -85,B 0,C 180,E1 -25958.556,E2 -25958.556} C_VEL
LIN {X 0,Y 150.447,Z 283.44,A -85,B 0,C 180,E1 -25959.451,E2 -25959.451} C_VEL
LIN {X 0,Y 147.363,Z 297.672,A -85,B 0,C 180,E1 -25960.796,E2 -25960.796} C_VEL
LIN {X 0,Y 143.477,Z 311.785,A -85,B 0,C 180,E1 -25962.72,E2 -25962.72} C_VEL
LIN {X 0,Y 139.168,Z 324.374,A -85,B 0,C 180,E1 -25965.015,E2 -25965.015} C_VEL
LIN {X 0,Y 135.708,Z 333.591,A -85,B 0,C 180,E1 -25967.215,E2 -25967.215} C_VEL
LIN {X 0,Y 132.769,Z 340.324,A -85,B 0,C 180,E1 -25969.082,E2 -25969.082} C_VEL
LIN {X 0,Y 127.924,Z 351.046,A -85,B 0,C 180,E1 -25972.825,E2 -25972.825} C_VEL
LIN {X 0,Y 123.351,Z 360.711,A -85,B 0,C 180,E1 -25977.236,E2 -25977.236} C_VEL
LIN {X 0,Y 119.05,Z 369.635,A -85,B 0,C 180,E1 -25982.573,E2 -25982.573} C_VEL
LIN {X 0,Y 116.506,Z 375.313,A -85,B 0,C 180,E1 -25986.92,E2 -25986.92} C_VEL
LIN {X 0,Y 114.262,Z 380.775,A -85,B 0,C 180,E1 -25992.094,E2 -25992.094} C_VEL
LIN {X 0,Y 112.647,Z 386.497,A -85,B 0,C 180,E1 -25999.218,E2 -25999.218} C_VEL
LIN {X 0,Y 112.266,Z 388.736,A -85,B 0,C 180,E1 -26002.813,E2 -26002.813} C_VEL
LIN {X 0,Y 112.145,Z 390.587,A -85,B 0,C 180,E1 -26006.412,E2 -26006.412} C_VEL
LIN {X 0,Y 112.28,Z 392.068,A -85,B 0,C 180,E1 -26010.005,E2 -26010.005} C_VEL
LIN {X 0,Y 112.211,Z 393.17,A -85,B 0,C 180,E1 -26013.596,E2 -26013.596} C_VEL
LIN {X 0,Y 112.708,Z 394.353,A -85,B 0,C 180,E1 -26020.787,E2 -26020.787} C_VEL
LIN {X 0,Y 114.567,Z 394.236,A -85,B 0,C 180,E1 -26027.867,E2 -26027.867} C_VEL
LIN {X 0,Y 118.352,Z 392.722,A -85,B 0,C 180,E1 -26034.929,E2 -26034.929} C_VEL
LIN {X 0,Y 119.644,Z 391.785,A -85,B 0,C 180,E1 -26037.663,E2 -26037.663} C_VEL
LIN {X 0,Y 120.619,Z 389.846,A -85,B 0,C 180,E1 -26042.288,E2 -26042.288} C_VEL
LIN {X 0,Y 122.302,Z 387.468,A -85,B 0,C 180,E1 -26046.756,E2 -26046.756} C_VEL
LIN {X 0,Y 124.609,Z 385.666,A -85,B 0,C 180,E1 -26049.134,E2 -26049.134} C_VEL
LIN {X 0,Y 131.985,Z 380.633,A -85,B 0,C 180,E1 -26053.813,E2 -26053.813} C_VEL
LIN {X 0,Y 138.717,Z 375.462,A -85,B 0,C 180,E1 -26057.282,E2 -26057.282} C_VEL
LIN {X 0,Y 147.255,Z 368.038,A -85,B 0,C 180,E1 -26060.861,E2 -26060.861} C_VEL
LIN {X 0,Y 154.943,Z 360.342,A -85,B 0,C 180,E1 -26063.622,E2 -26063.622} C_VEL
LIN {X 0,Y 162.956,Z 351.108,A -85,B 0,C 180,E1 -26066.127,E2 -26066.127} C_VEL
LIN {X 0,Y 171.351,Z 339.873,A -85,B 0,C 180,E1 -26068.333,E2 -26068.333} C_VEL
LIN {X 0,Y 178.515,Z 328.488,A -85,B 0,C 180,E1 -26070.017,E2 -26070.017} C_VEL
LIN {X 0,Y 185.163,Z 315.887,A -85,B 0,C 180,E1 -26071.375,E2 -26071.375} C_VEL
LIN {X 0,Y 190.396,Z 303.666,A -85,B 0,C 180,E1 -26072.368,E2 -26072.368} C_VEL
LIN {X 0,Y 194.939,Z 290.195,A -85,B 0,C 180,E1 -26073.169,E2 -26073.169} C_VEL
LIN {X 0,Y 198.357,Z 276.415,A -85,B 0,C 180,E1 -26073.738,E2 -26073.738} C_VEL
LIN {X 0,Y 200.495,Z 262.877,A -85,B 0,C 180,E1 -26074.147,E2 -26074.147} C_VEL
LIN {X 0,Y 201.808,Z 250.377,A -85,B 0,C 180,E1 -26074.464,E2 -26074.464} C_VEL
LIN {X 0,Y 200.814,Z 246.932,A -85,B 0,C 180,E1 -26075.746,E2 -26075.746} C_VEL
LIN {X 0,Y 198.723,Z 240.756,A -85,B 0,C 180,E1 -26078.701,E2 -26078.701} C_VEL
LIN {X 0,Y 196.795,Z 235.616,A -85,B 0,C 180,E1 -26082.188,E2 -26082.188} C_VEL
LIN {X 0,Y 195.601,Z 232.865,A -85,B 0,C 180,E1 -26085.1,E2 -26085.1} C_VEL
LIN {X 0,Y 194.429,Z 229.556,A -85,B 0,C 180,E1 -26091.68,E2 -26091.68} C_VEL
LIN {X 0,Y 194.547,Z 229.624,A -85,B 0,C 180,E1 -26094.202,E2 -26094.202} C_VEL
LIN {X 0,Y 196.033,Z 233.357,A -85,B 0,C 180,E1 -26100.365,E2 -26100.365} C_VEL
LIN {X 0,Y 197.595,Z 236.847,A -85,B 0,C 180,E1 -26103.662,E2 -26103.662} C_VEL
LIN {X 0,Y 199.557,Z 241.091,A -85,B 0,C 180,E1 -26106.685,E2 -26106.685} C_VEL
LIN {X 0,Y 202.152,Z 246.8,A -85,B 0,C 180,E1 -26109.846,E2 -26109.846} C_VEL
LIN {X 0,Y 199.704,Z 267.273,A -85,B 0,C 180,E1 -26110.383,E2 -26110.383} C_VEL
LIN {X 0,Y 196.668,Z 281.741,A -85,B 0,C 180,E1 -26110.959,E2 -26110.959} C_VEL
LIN {X 0,Y 192.873,Z 294.454,A -85,B 0,C 180,E1 -26111.67,E2 -26111.67} C_VEL
LIN {X 0,Y 188.194,Z 306.806,A -85,B 0,C 180,E1 -26112.665,E2 -26112.665} C_VEL
LIN {X 0,Y 182.525,Z 318.843,A -85,B 0,C 180,E1 -26113.931,E2 -26113.931} C_VEL
LIN {X 0,Y 175.952,Z 330.343,A -85,B 0,C 180,E1 -26115.492,E2 -26115.492} C_VEL
LIN {X 0,Y 168.508,Z 341.271,A -85,B 0,C 180,E1 -26117.426,E2 -26117.426} C_VEL
LIN {X 0,Y 160.581,Z 351.203,A -85,B 0,C 180,E1 -26119.775,E2 -26119.775} C_VEL
LIN {X 0,Y 152.255,Z 360.132,A -85,B 0,C 180,E1 -26122.595,E2 -26122.595} C_VEL
LIN {X 0,Y 143.364,Z 368.306,A -85,B 0,C 180,E1 -26126.169,E2 -26126.169} C_VEL
LIN {X 0,Y 134.589,Z 375.233,A -85,B 0,C 180,E1 -26130.495,E2 -26130.495} C_VEL
LIN {X 0,Y 127.963,Z 379.79,A -85,B 0,C 180,E1 -26134.522,E2 -26134.522} C_VEL
LIN {X 0,Y 120.177,Z 384.295,A -85,B 0,C 180,E1 -26140.507,E2 -26140.507} C_VEL
LIN {X 0,Y 113.872,Z 387.214,A -85,B 0,C 180,E1 -26147.235,E2 -26147.235} C_VEL
LIN {X 0,Y 109.155,Z 388.637,A -85,B 0,C 180,E1 -26154.581,E2 -26154.581} C_VEL
LIN {X 0,Y 106.146,Z 388.594,A -85,B 0,C 180,E1 -26162.383,E2 -26162.383} C_VEL
LIN {X 0,Y 104.812,Z 387.085,A -85,B 0,C 180,E1 -26170.406,E2 -26170.406} C_VEL
LIN {X 0,Y 104.715,Z 384.16,A -85,B 0,C 180,E1 -26178.379,E2 -26178.379} C_VEL
LIN {X 0,Y 105.794,Z 380.535,A -85,B 0,C 180,E1 -26185.014,E2 -26185.014} C_VEL
LIN {X 0,Y 107.706,Z 375.422,A -85,B 0,C 180,E1 -26191.864,E2 -26191.864} C_VEL
LIN {X 0,Y 110.637,Z 369.105,A -85,B 0,C 180,E1 -26198.212,E2 -26198.212} C_VEL
LIN {X 0,Y 114.685,Z 361.234,A -85,B 0,C 180,E1 -26204.184,E2 -26204.184} C_VEL
LIN {X 0,Y 119.067,Z 352.765,A -85,B 0,C 180,E1 -26209.09,E2 -26209.09} C_VEL
LIN {X 0,Y 122.91,Z 344.93,A -85,B 0,C 180,E1 -26212.698,E2 -26212.698} C_VEL
LIN {X 0,Y 127.264,Z 335.4,A -85,B 0,C 180,E1 -26216.213,E2 -26216.213} C_VEL
